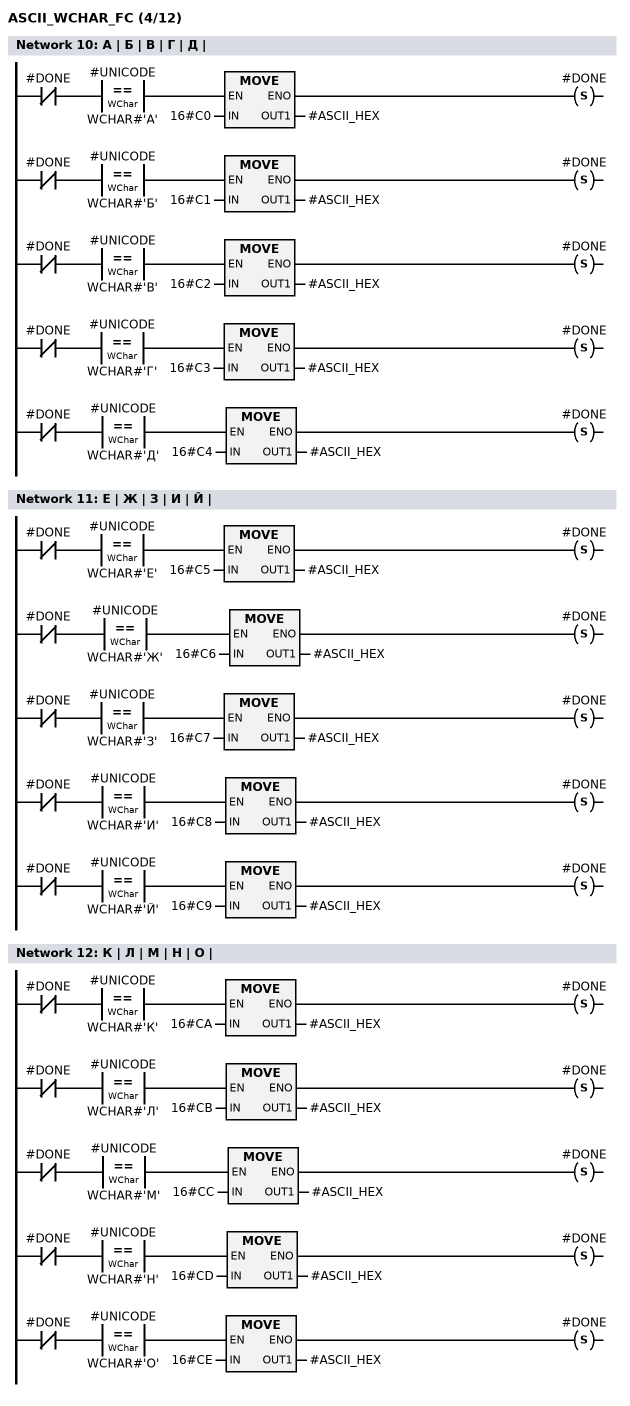
   RUNG wire#powerrail
      I_Contact( #DONE )
      { S7_Templates := "SrcType := WChar" } EQ_Contact(in1 := #UNICODE, in2 := WCHAR#'А')
      Move(in := 16#C0, out1 => #ASCII_HEX)
      S_Coil( #DONE )
   END_RUNG
   RUNG wire#powerrail
      I_Contact( #DONE )
      { S7_Templates := "SrcType := WChar" } EQ_Contact(in1 := #UNICODE, in2 := WCHAR#'Б')
      Move(in := 16#C1, out1 => #ASCII_HEX)
      S_Coil( #DONE )
   END_RUNG
   RUNG wire#powerrail
      I_Contact( #DONE )
      { S7_Templates := "SrcType := WChar" } EQ_Contact(in1 := #UNICODE, in2 := WCHAR#'В')
      Move(in := 16#C2, out1 => #ASCII_HEX)
      S_Coil( #DONE )
   END_RUNG
   RUNG wire#powerrail
      I_Contact( #DONE )
      { S7_Templates := "SrcType := WChar" } EQ_Contact(in1 := #UNICODE, in2 := WCHAR#'Г')
      Move(in := 16#C3, out1 => #ASCII_HEX)
      S_Coil( #DONE )
   END_RUNG
   RUNG wire#powerrail
      I_Contact( #DONE )
      { S7_Templates := "SrcType := WChar" } EQ_Contact(in1 := #UNICODE, in2 := WCHAR#'Д')
      Move(in := 16#C4, out1 => #ASCII_HEX)
      S_Coil( #DONE )
   END_RUNG
   // the same network as SCL:
   IF NOT #DONE AND (#UNICODE = WCHAR#'А') THEN
       #ASCII_HEX := 16#C0;
       #DONE := TRUE;
   END_IF;
   IF NOT #DONE AND (#UNICODE = WCHAR#'Б') THEN
       #ASCII_HEX := 16#C1;
       #DONE := TRUE;
   END_IF;
   IF NOT #DONE AND (#UNICODE = WCHAR#'В') THEN
       #ASCII_HEX := 16#C2;
       #DONE := TRUE;
   END_IF;
   IF NOT #DONE AND (#UNICODE = WCHAR#'Г') THEN
       #ASCII_HEX := 16#C3;
       #DONE := TRUE;
   END_IF;
   IF NOT #DONE AND (#UNICODE = WCHAR#'Д') THEN
       #ASCII_HEX := 16#C4;
       #DONE := TRUE;
   END_IF;
END_REGION

REGION Network 11: Е | Ж | З | И | Й |
   RUNG wire#powerrail
      I_Contact( #DONE )
      { S7_Templates := "SrcType := WChar" } EQ_Contact(in1 := #UNICODE, in2 := WCHAR#'Е')
      Move(in := 16#C5, out1 => #ASCII_HEX)
      S_Coil( #DONE )
   END_RUNG
   RUNG wire#powerrail
      I_Contact( #DONE )
      { S7_Templates := "SrcType := WChar" } EQ_Contact(in1 := #UNICODE, in2 := WCHAR#'Ж')
      Move(in := 16#C6, out1 => #ASCII_HEX)
      S_Coil( #DONE )
   END_RUNG
   RUNG wire#powerrail
      I_Contact( #DONE )
      { S7_Templates := "SrcType := WChar" } EQ_Contact(in1 := #UNICODE, in2 := WCHAR#'З')
      Move(in := 16#C7, out1 => #ASCII_HEX)
      S_Coil( #DONE )
   END_RUNG
   RUNG wire#powerrail
      I_Contact( #DONE )
      { S7_Templates := "SrcType := WChar" } EQ_Contact(in1 := #UNICODE, in2 := WCHAR#'И')
      Move(in := 16#C8, out1 => #ASCII_HEX)
      S_Coil( #DONE )
   END_RUNG
   RUNG wire#powerrail
      I_Contact( #DONE )
      { S7_Templates := "SrcType := WChar" } EQ_Contact(in1 := #UNICODE, in2 := WCHAR#'Й')
      Move(in := 16#C9, out1 => #ASCII_HEX)
      S_Coil( #DONE )
   END_RUNG
   // the same network as SCL:
   IF NOT #DONE AND (#UNICODE = WCHAR#'Е') THEN
       #ASCII_HEX := 16#C5;
       #DONE := TRUE;
   END_IF;
   IF NOT #DONE AND (#UNICODE = WCHAR#'Ж') THEN
       #ASCII_HEX := 16#C6;
       #DONE := TRUE;
   END_IF;
   IF NOT #DONE AND (#UNICODE = WCHAR#'З') THEN
       #ASCII_HEX := 16#C7;
       #DONE := TRUE;
   END_IF;
   IF NOT #DONE AND (#UNICODE = WCHAR#'И') THEN
       #ASCII_HEX := 16#C8;
       #DONE := TRUE;
   END_IF;
   IF NOT #DONE AND (#UNICODE = WCHAR#'Й') THEN
       #ASCII_HEX := 16#C9;
       #DONE := TRUE;
   END_IF;
END_REGION

REGION Network 12: К | Л | М | Н | О |
   RUNG wire#powerrail
      I_Contact( #DONE )
      { S7_Templates := "SrcType := WChar" } EQ_Contact(in1 := #UNICODE, in2 := WCHAR#'К')
      Move(in := 16#CA, out1 => #ASCII_HEX)
      S_Coil( #DONE )
   END_RUNG
   RUNG wire#powerrail
      I_Contact( #DONE )
      { S7_Templates := "SrcType := WChar" } EQ_Contact(in1 := #UNICODE, in2 := WCHAR#'Л')
      Move(in := 16#CB, out1 => #ASCII_HEX)
      S_Coil( #DONE )
   END_RUNG
   RUNG wire#powerrail
      I_Contact( #DONE )
      { S7_Templates := "SrcType := WChar" } EQ_Contact(in1 := #UNICODE, in2 := WCHAR#'М')
      Move(in := 16#CC, out1 => #ASCII_HEX)
      S_Coil( #DONE )
   END_RUNG
   RUNG wire#powerrail
      I_Contact( #DONE )
      { S7_Templates := "SrcType := WChar" } EQ_Contact(in1 := #UNICODE, in2 := WCHAR#'Н')
      Move(in := 16#CD, out1 => #ASCII_HEX)
      S_Coil( #DONE )
   END_RUNG
   RUNG wire#powerrail
      I_Contact( #DONE )
      { S7_Templates := "SrcType := WChar" } EQ_Contact(in1 := #UNICODE, in2 := WCHAR#'О')
      Move(in := 16#CE, out1 => #ASCII_HEX)
      S_Coil( #DONE )
   END_RUNG
   // the same network as SCL:
   IF NOT #DONE AND (#UNICODE = WCHAR#'К') THEN
       #ASCII_HEX := 16#CA;
       #DONE := TRUE;
   END_IF;
   IF NOT #DONE AND (#UNICODE = WCHAR#'Л') THEN
       #ASCII_HEX := 16#CB;
       #DONE := TRUE;
   END_IF;
   IF NOT #DONE AND (#UNICODE = WCHAR#'М') THEN
       #ASCII_HEX := 16#CC;
       #DONE := TRUE;
   END_IF;
   IF NOT #DONE AND (#UNICODE = WCHAR#'Н') THEN
       #ASCII_HEX := 16#CD;
       #DONE := TRUE;
   END_IF;
   IF NOT #DONE AND (#UNICODE = WCHAR#'О') THEN
       #ASCII_HEX := 16#CE;
       #DONE := TRUE;
   END_IF;
END_REGION

REGION Network 13: П | Р | С | Т | У |
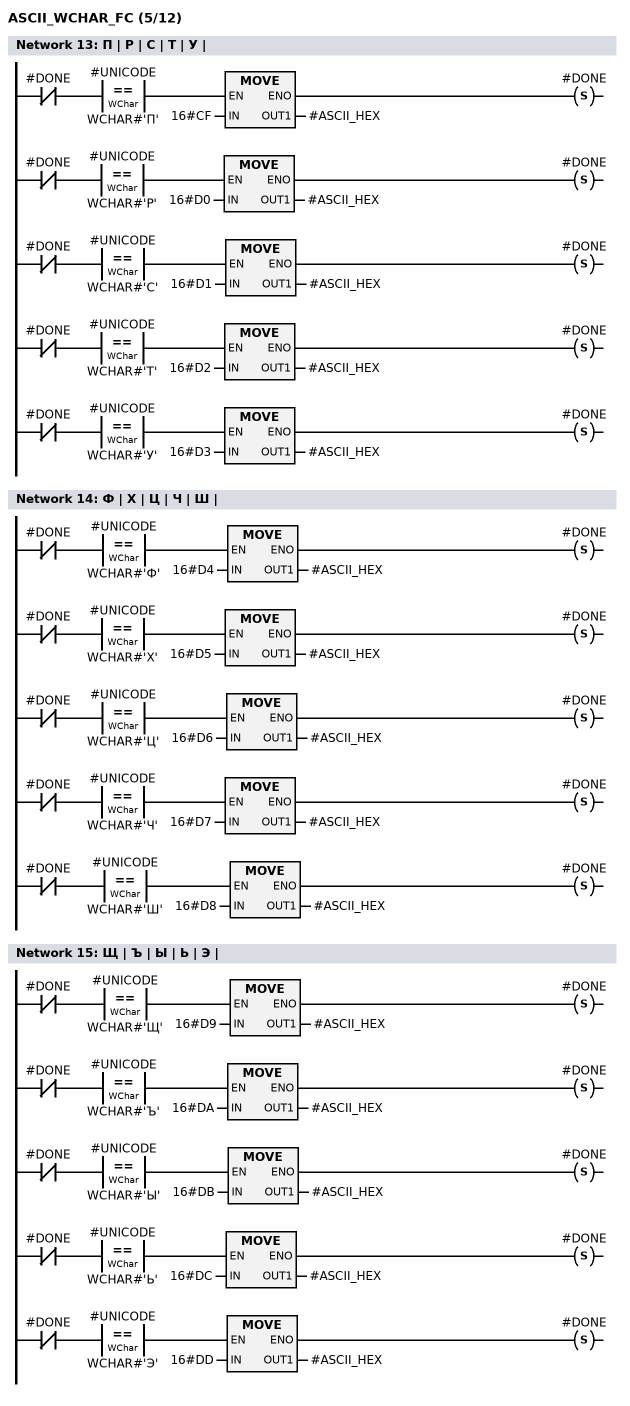
   RUNG wire#powerrail
      I_Contact( #DONE )
      { S7_Templates := "SrcType := WChar" } EQ_Contact(in1 := #UNICODE, in2 := WCHAR#'П')
      Move(in := 16#CF, out1 => #ASCII_HEX)
      S_Coil( #DONE )
   END_RUNG
   RUNG wire#powerrail
      I_Contact( #DONE )
      { S7_Templates := "SrcType := WChar" } EQ_Contact(in1 := #UNICODE, in2 := WCHAR#'Р')
      Move(in := 16#D0, out1 => #ASCII_HEX)
      S_Coil( #DONE )
   END_RUNG
   RUNG wire#powerrail
      I_Contact( #DONE )
      { S7_Templates := "SrcType := WChar" } EQ_Contact(in1 := #UNICODE, in2 := WCHAR#'С')
      Move(in := 16#D1, out1 => #ASCII_HEX)
      S_Coil( #DONE )
   END_RUNG
   RUNG wire#powerrail
      I_Contact( #DONE )
      { S7_Templates := "SrcType := WChar" } EQ_Contact(in1 := #UNICODE, in2 := WCHAR#'Т')
      Move(in := 16#D2, out1 => #ASCII_HEX)
      S_Coil( #DONE )
   END_RUNG
   RUNG wire#powerrail
      I_Contact( #DONE )
      { S7_Templates := "SrcType := WChar" } EQ_Contact(in1 := #UNICODE, in2 := WCHAR#'У')
      Move(in := 16#D3, out1 => #ASCII_HEX)
      S_Coil( #DONE )
   END_RUNG
   // the same network as SCL:
   IF NOT #DONE AND (#UNICODE = WCHAR#'П') THEN
       #ASCII_HEX := 16#CF;
       #DONE := TRUE;
   END_IF;
   IF NOT #DONE AND (#UNICODE = WCHAR#'Р') THEN
       #ASCII_HEX := 16#D0;
       #DONE := TRUE;
   END_IF;
   IF NOT #DONE AND (#UNICODE = WCHAR#'С') THEN
       #ASCII_HEX := 16#D1;
       #DONE := TRUE;
   END_IF;
   IF NOT #DONE AND (#UNICODE = WCHAR#'Т') THEN
       #ASCII_HEX := 16#D2;
       #DONE := TRUE;
   END_IF;
   IF NOT #DONE AND (#UNICODE = WCHAR#'У') THEN
       #ASCII_HEX := 16#D3;
       #DONE := TRUE;
   END_IF;
END_REGION

REGION Network 14: Ф | Х | Ц | Ч | Ш |
   RUNG wire#powerrail
      I_Contact( #DONE )
      { S7_Templates := "SrcType := WChar" } EQ_Contact(in1 := #UNICODE, in2 := WCHAR#'Ф')
      Move(in := 16#D4, out1 => #ASCII_HEX)
      S_Coil( #DONE )
   END_RUNG
   RUNG wire#powerrail
      I_Contact( #DONE )
      { S7_Templates := "SrcType := WChar" } EQ_Contact(in1 := #UNICODE, in2 := WCHAR#'Х')
      Move(in := 16#D5, out1 => #ASCII_HEX)
      S_Coil( #DONE )
   END_RUNG
   RUNG wire#powerrail
      I_Contact( #DONE )
      { S7_Templates := "SrcType := WChar" } EQ_Contact(in1 := #UNICODE, in2 := WCHAR#'Ц')
      Move(in := 16#D6, out1 => #ASCII_HEX)
      S_Coil( #DONE )
   END_RUNG
   RUNG wire#powerrail
      I_Contact( #DONE )
      { S7_Templates := "SrcType := WChar" } EQ_Contact(in1 := #UNICODE, in2 := WCHAR#'Ч')
      Move(in := 16#D7, out1 => #ASCII_HEX)
      S_Coil( #DONE )
   END_RUNG
   RUNG wire#powerrail
      I_Contact( #DONE )
      { S7_Templates := "SrcType := WChar" } EQ_Contact(in1 := #UNICODE, in2 := WCHAR#'Ш')
      Move(in := 16#D8, out1 => #ASCII_HEX)
      S_Coil( #DONE )
   END_RUNG
   // the same network as SCL:
   IF NOT #DONE AND (#UNICODE = WCHAR#'Ф') THEN
       #ASCII_HEX := 16#D4;
       #DONE := TRUE;
   END_IF;
   IF NOT #DONE AND (#UNICODE = WCHAR#'Х') THEN
       #ASCII_HEX := 16#D5;
       #DONE := TRUE;
   END_IF;
   IF NOT #DONE AND (#UNICODE = WCHAR#'Ц') THEN
       #ASCII_HEX := 16#D6;
       #DONE := TRUE;
   END_IF;
   IF NOT #DONE AND (#UNICODE = WCHAR#'Ч') THEN
       #ASCII_HEX := 16#D7;
       #DONE := TRUE;
   END_IF;
   IF NOT #DONE AND (#UNICODE = WCHAR#'Ш') THEN
       #ASCII_HEX := 16#D8;
       #DONE := TRUE;
   END_IF;
END_REGION

REGION Network 15: Щ | Ъ | Ы | Ь | Э |
   RUNG wire#powerrail
      I_Contact( #DONE )
      { S7_Templates := "SrcType := WChar" } EQ_Contact(in1 := #UNICODE, in2 := WCHAR#'Щ')
      Move(in := 16#D9, out1 => #ASCII_HEX)
      S_Coil( #DONE )
   END_RUNG
   RUNG wire#powerrail
      I_Contact( #DONE )
      { S7_Templates := "SrcType := WChar" } EQ_Contact(in1 := #UNICODE, in2 := WCHAR#'Ъ')
      Move(in := 16#DA, out1 => #ASCII_HEX)
      S_Coil( #DONE )
   END_RUNG
   RUNG wire#powerrail
      I_Contact( #DONE )
      { S7_Templates := "SrcType := WChar" } EQ_Contact(in1 := #UNICODE, in2 := WCHAR#'Ы')
      Move(in := 16#DB, out1 => #ASCII_HEX)
      S_Coil( #DONE )
   END_RUNG
   RUNG wire#powerrail
      I_Contact( #DONE )
      { S7_Templates := "SrcType := WChar" } EQ_Contact(in1 := #UNICODE, in2 := WCHAR#'Ь')
      Move(in := 16#DC, out1 => #ASCII_HEX)
      S_Coil( #DONE )
   END_RUNG
   RUNG wire#powerrail
      I_Contact( #DONE )
      { S7_Templates := "SrcType := WChar" } EQ_Contact(in1 := #UNICODE, in2 := WCHAR#'Э')
      Move(in := 16#DD, out1 => #ASCII_HEX)
      S_Coil( #DONE )
   END_RUNG
   // the same network as SCL:
   IF NOT #DONE AND (#UNICODE = WCHAR#'Щ') THEN
       #ASCII_HEX := 16#D9;
       #DONE := TRUE;
   END_IF;
   IF NOT #DONE AND (#UNICODE = WCHAR#'Ъ') THEN
       #ASCII_HEX := 16#DA;
       #DONE := TRUE;
   END_IF;
   IF NOT #DONE AND (#UNICODE = WCHAR#'Ы') THEN
       #ASCII_HEX := 16#DB;
       #DONE := TRUE;
   END_IF;
   IF NOT #DONE AND (#UNICODE = WCHAR#'Ь') THEN
       #ASCII_HEX := 16#DC;
       #DONE := TRUE;
   END_IF;
   IF NOT #DONE AND (#UNICODE = WCHAR#'Э') THEN
       #ASCII_HEX := 16#DD;
       #DONE := TRUE;
   END_IF;
END_REGION

REGION Network 16: Ю | Я |
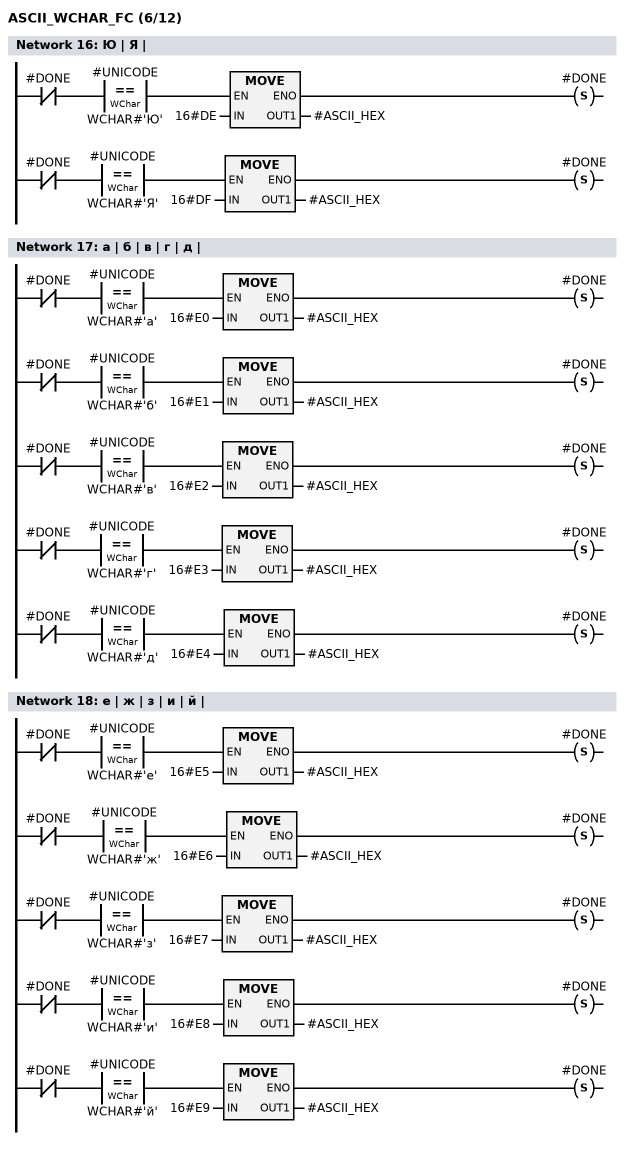
   RUNG wire#powerrail
      I_Contact( #DONE )
      { S7_Templates := "SrcType := WChar" } EQ_Contact(in1 := #UNICODE, in2 := WCHAR#'Ю')
      Move(in := 16#DE, out1 => #ASCII_HEX)
      S_Coil( #DONE )
   END_RUNG
   RUNG wire#powerrail
      I_Contact( #DONE )
      { S7_Templates := "SrcType := WChar" } EQ_Contact(in1 := #UNICODE, in2 := WCHAR#'Я')
      Move(in := 16#DF, out1 => #ASCII_HEX)
      S_Coil( #DONE )
   END_RUNG
   // the same network as SCL:
   IF NOT #DONE AND (#UNICODE = WCHAR#'Ю') THEN
       #ASCII_HEX := 16#DE;
       #DONE := TRUE;
   END_IF;
   IF NOT #DONE AND (#UNICODE = WCHAR#'Я') THEN
       #ASCII_HEX := 16#DF;
       #DONE := TRUE;
   END_IF;
END_REGION

REGION Network 17: а | б | в | г | д |
   RUNG wire#powerrail
      I_Contact( #DONE )
      { S7_Templates := "SrcType := WChar" } EQ_Contact(in1 := #UNICODE, in2 := WCHAR#'а')
      Move(in := 16#E0, out1 => #ASCII_HEX)
      S_Coil( #DONE )
   END_RUNG
   RUNG wire#powerrail
      I_Contact( #DONE )
      { S7_Templates := "SrcType := WChar" } EQ_Contact(in1 := #UNICODE, in2 := WCHAR#'б')
      Move(in := 16#E1, out1 => #ASCII_HEX)
      S_Coil( #DONE )
   END_RUNG
   RUNG wire#powerrail
      I_Contact( #DONE )
      { S7_Templates := "SrcType := WChar" } EQ_Contact(in1 := #UNICODE, in2 := WCHAR#'в')
      Move(in := 16#E2, out1 => #ASCII_HEX)
      S_Coil( #DONE )
   END_RUNG
   RUNG wire#powerrail
      I_Contact( #DONE )
      { S7_Templates := "SrcType := WChar" } EQ_Contact(in1 := #UNICODE, in2 := WCHAR#'г')
      Move(in := 16#E3, out1 => #ASCII_HEX)
      S_Coil( #DONE )
   END_RUNG
   RUNG wire#powerrail
      I_Contact( #DONE )
      { S7_Templates := "SrcType := WChar" } EQ_Contact(in1 := #UNICODE, in2 := WCHAR#'д')
      Move(in := 16#E4, out1 => #ASCII_HEX)
      S_Coil( #DONE )
   END_RUNG
   // the same network as SCL:
   IF NOT #DONE AND (#UNICODE = WCHAR#'а') THEN
       #ASCII_HEX := 16#E0;
       #DONE := TRUE;
   END_IF;
   IF NOT #DONE AND (#UNICODE = WCHAR#'б') THEN
       #ASCII_HEX := 16#E1;
       #DONE := TRUE;
   END_IF;
   IF NOT #DONE AND (#UNICODE = WCHAR#'в') THEN
       #ASCII_HEX := 16#E2;
       #DONE := TRUE;
   END_IF;
   IF NOT #DONE AND (#UNICODE = WCHAR#'г') THEN
       #ASCII_HEX := 16#E3;
       #DONE := TRUE;
   END_IF;
   IF NOT #DONE AND (#UNICODE = WCHAR#'д') THEN
       #ASCII_HEX := 16#E4;
       #DONE := TRUE;
   END_IF;
END_REGION

REGION Network 18: е | ж | з | и | й |
   RUNG wire#powerrail
      I_Contact( #DONE )
      { S7_Templates := "SrcType := WChar" } EQ_Contact(in1 := #UNICODE, in2 := WCHAR#'е')
      Move(in := 16#E5, out1 => #ASCII_HEX)
      S_Coil( #DONE )
   END_RUNG
   RUNG wire#powerrail
      I_Contact( #DONE )
      { S7_Templates := "SrcType := WChar" } EQ_Contact(in1 := #UNICODE, in2 := WCHAR#'ж')
      Move(in := 16#E6, out1 => #ASCII_HEX)
      S_Coil( #DONE )
   END_RUNG
   RUNG wire#powerrail
      I_Contact( #DONE )
      { S7_Templates := "SrcType := WChar" } EQ_Contact(in1 := #UNICODE, in2 := WCHAR#'з')
      Move(in := 16#E7, out1 => #ASCII_HEX)
      S_Coil( #DONE )
   END_RUNG
   RUNG wire#powerrail
      I_Contact( #DONE )
      { S7_Templates := "SrcType := WChar" } EQ_Contact(in1 := #UNICODE, in2 := WCHAR#'и')
      Move(in := 16#E8, out1 => #ASCII_HEX)
      S_Coil( #DONE )
   END_RUNG
   RUNG wire#powerrail
      I_Contact( #DONE )
      { S7_Templates := "SrcType := WChar" } EQ_Contact(in1 := #UNICODE, in2 := WCHAR#'й')
      Move(in := 16#E9, out1 => #ASCII_HEX)
      S_Coil( #DONE )
   END_RUNG
   // the same network as SCL:
   IF NOT #DONE AND (#UNICODE = WCHAR#'е') THEN
       #ASCII_HEX := 16#E5;
       #DONE := TRUE;
   END_IF;
   IF NOT #DONE AND (#UNICODE = WCHAR#'ж') THEN
       #ASCII_HEX := 16#E6;
       #DONE := TRUE;
   END_IF;
   IF NOT #DONE AND (#UNICODE = WCHAR#'з') THEN
       #ASCII_HEX := 16#E7;
       #DONE := TRUE;
   END_IF;
   IF NOT #DONE AND (#UNICODE = WCHAR#'и') THEN
       #ASCII_HEX := 16#E8;
       #DONE := TRUE;
   END_IF;
   IF NOT #DONE AND (#UNICODE = WCHAR#'й') THEN
       #ASCII_HEX := 16#E9;
       #DONE := TRUE;
   END_IF;
END_REGION

REGION Network 19: к | л | м | н | о |
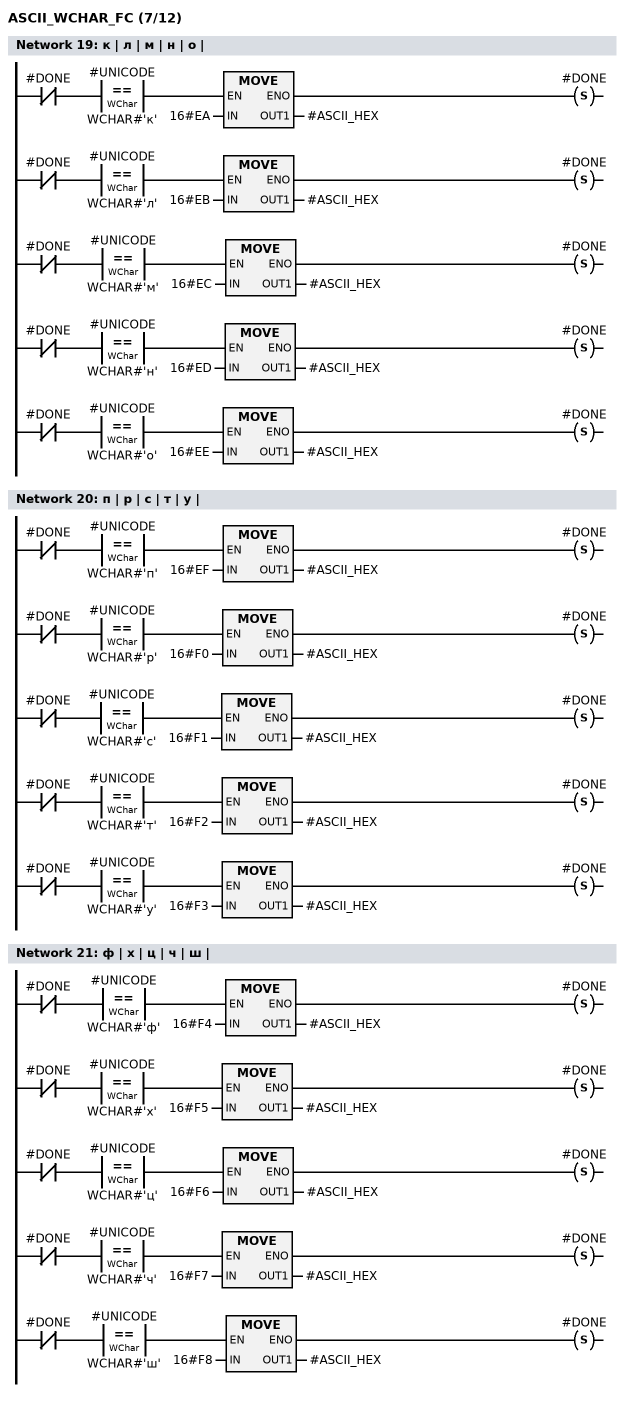
   RUNG wire#powerrail
      I_Contact( #DONE )
      { S7_Templates := "SrcType := WChar" } EQ_Contact(in1 := #UNICODE, in2 := WCHAR#'к')
      Move(in := 16#EA, out1 => #ASCII_HEX)
      S_Coil( #DONE )
   END_RUNG
   RUNG wire#powerrail
      I_Contact( #DONE )
      { S7_Templates := "SrcType := WChar" } EQ_Contact(in1 := #UNICODE, in2 := WCHAR#'л')
      Move(in := 16#EB, out1 => #ASCII_HEX)
      S_Coil( #DONE )
   END_RUNG
   RUNG wire#powerrail
      I_Contact( #DONE )
      { S7_Templates := "SrcType := WChar" } EQ_Contact(in1 := #UNICODE, in2 := WCHAR#'м')
      Move(in := 16#EC, out1 => #ASCII_HEX)
      S_Coil( #DONE )
   END_RUNG
   RUNG wire#powerrail
      I_Contact( #DONE )
      { S7_Templates := "SrcType := WChar" } EQ_Contact(in1 := #UNICODE, in2 := WCHAR#'н')
      Move(in := 16#ED, out1 => #ASCII_HEX)
      S_Coil( #DONE )
   END_RUNG
   RUNG wire#powerrail
      I_Contact( #DONE )
      { S7_Templates := "SrcType := WChar" } EQ_Contact(in1 := #UNICODE, in2 := WCHAR#'о')
      Move(in := 16#EE, out1 => #ASCII_HEX)
      S_Coil( #DONE )
   END_RUNG
   // the same network as SCL:
   IF NOT #DONE AND (#UNICODE = WCHAR#'к') THEN
       #ASCII_HEX := 16#EA;
       #DONE := TRUE;
   END_IF;
   IF NOT #DONE AND (#UNICODE = WCHAR#'л') THEN
       #ASCII_HEX := 16#EB;
       #DONE := TRUE;
   END_IF;
   IF NOT #DONE AND (#UNICODE = WCHAR#'м') THEN
       #ASCII_HEX := 16#EC;
       #DONE := TRUE;
   END_IF;
   IF NOT #DONE AND (#UNICODE = WCHAR#'н') THEN
       #ASCII_HEX := 16#ED;
       #DONE := TRUE;
   END_IF;
   IF NOT #DONE AND (#UNICODE = WCHAR#'о') THEN
       #ASCII_HEX := 16#EE;
       #DONE := TRUE;
   END_IF;
END_REGION

REGION Network 20: п | р | с | т | у |
   RUNG wire#powerrail
      I_Contact( #DONE )
      { S7_Templates := "SrcType := WChar" } EQ_Contact(in1 := #UNICODE, in2 := WCHAR#'п')
      Move(in := 16#EF, out1 => #ASCII_HEX)
      S_Coil( #DONE )
   END_RUNG
   RUNG wire#powerrail
      I_Contact( #DONE )
      { S7_Templates := "SrcType := WChar" } EQ_Contact(in1 := #UNICODE, in2 := WCHAR#'р')
      Move(in := 16#F0, out1 => #ASCII_HEX)
      S_Coil( #DONE )
   END_RUNG
   RUNG wire#powerrail
      I_Contact( #DONE )
      { S7_Templates := "SrcType := WChar" } EQ_Contact(in1 := #UNICODE, in2 := WCHAR#'с')
      Move(in := 16#F1, out1 => #ASCII_HEX)
      S_Coil( #DONE )
   END_RUNG
   RUNG wire#powerrail
      I_Contact( #DONE )
      { S7_Templates := "SrcType := WChar" } EQ_Contact(in1 := #UNICODE, in2 := WCHAR#'т')
      Move(in := 16#F2, out1 => #ASCII_HEX)
      S_Coil( #DONE )
   END_RUNG
   RUNG wire#powerrail
      I_Contact( #DONE )
      { S7_Templates := "SrcType := WChar" } EQ_Contact(in1 := #UNICODE, in2 := WCHAR#'у')
      Move(in := 16#F3, out1 => #ASCII_HEX)
      S_Coil( #DONE )
   END_RUNG
   // the same network as SCL:
   IF NOT #DONE AND (#UNICODE = WCHAR#'п') THEN
       #ASCII_HEX := 16#EF;
       #DONE := TRUE;
   END_IF;
   IF NOT #DONE AND (#UNICODE = WCHAR#'р') THEN
       #ASCII_HEX := 16#F0;
       #DONE := TRUE;
   END_IF;
   IF NOT #DONE AND (#UNICODE = WCHAR#'с') THEN
       #ASCII_HEX := 16#F1;
       #DONE := TRUE;
   END_IF;
   IF NOT #DONE AND (#UNICODE = WCHAR#'т') THEN
       #ASCII_HEX := 16#F2;
       #DONE := TRUE;
   END_IF;
   IF NOT #DONE AND (#UNICODE = WCHAR#'у') THEN
       #ASCII_HEX := 16#F3;
       #DONE := TRUE;
   END_IF;
END_REGION

REGION Network 21: ф | х | ц | ч | ш |
   RUNG wire#powerrail
      I_Contact( #DONE )
      { S7_Templates := "SrcType := WChar" } EQ_Contact(in1 := #UNICODE, in2 := WCHAR#'ф')
      Move(in := 16#F4, out1 => #ASCII_HEX)
      S_Coil( #DONE )
   END_RUNG
   RUNG wire#powerrail
      I_Contact( #DONE )
      { S7_Templates := "SrcType := WChar" } EQ_Contact(in1 := #UNICODE, in2 := WCHAR#'х')
      Move(in := 16#F5, out1 => #ASCII_HEX)
      S_Coil( #DONE )
   END_RUNG
   RUNG wire#powerrail
      I_Contact( #DONE )
      { S7_Templates := "SrcType := WChar" } EQ_Contact(in1 := #UNICODE, in2 := WCHAR#'ц')
      Move(in := 16#F6, out1 => #ASCII_HEX)
      S_Coil( #DONE )
   END_RUNG
   RUNG wire#powerrail
      I_Contact( #DONE )
      { S7_Templates := "SrcType := WChar" } EQ_Contact(in1 := #UNICODE, in2 := WCHAR#'ч')
      Move(in := 16#F7, out1 => #ASCII_HEX)
      S_Coil( #DONE )
   END_RUNG
   RUNG wire#powerrail
      I_Contact( #DONE )
      { S7_Templates := "SrcType := WChar" } EQ_Contact(in1 := #UNICODE, in2 := WCHAR#'ш')
      Move(in := 16#F8, out1 => #ASCII_HEX)
      S_Coil( #DONE )
   END_RUNG
   // the same network as SCL:
   IF NOT #DONE AND (#UNICODE = WCHAR#'ф') THEN
       #ASCII_HEX := 16#F4;
       #DONE := TRUE;
   END_IF;
   IF NOT #DONE AND (#UNICODE = WCHAR#'х') THEN
       #ASCII_HEX := 16#F5;
       #DONE := TRUE;
   END_IF;
   IF NOT #DONE AND (#UNICODE = WCHAR#'ц') THEN
       #ASCII_HEX := 16#F6;
       #DONE := TRUE;
   END_IF;
   IF NOT #DONE AND (#UNICODE = WCHAR#'ч') THEN
       #ASCII_HEX := 16#F7;
       #DONE := TRUE;
   END_IF;
   IF NOT #DONE AND (#UNICODE = WCHAR#'ш') THEN
       #ASCII_HEX := 16#F8;
       #DONE := TRUE;
   END_IF;
END_REGION

REGION Network 22: щ | ъ | ы | ь | э |
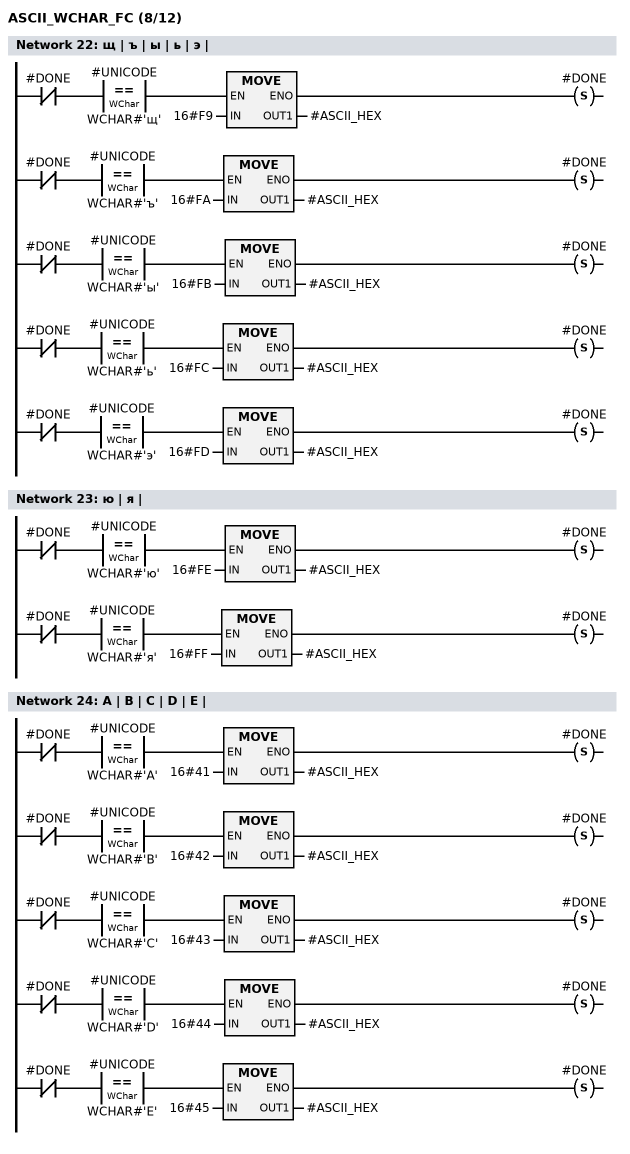
   RUNG wire#powerrail
      I_Contact( #DONE )
      { S7_Templates := "SrcType := WChar" } EQ_Contact(in1 := #UNICODE, in2 := WCHAR#'щ')
      Move(in := 16#F9, out1 => #ASCII_HEX)
      S_Coil( #DONE )
   END_RUNG
   RUNG wire#powerrail
      I_Contact( #DONE )
      { S7_Templates := "SrcType := WChar" } EQ_Contact(in1 := #UNICODE, in2 := WCHAR#'ъ')
      Move(in := 16#FA, out1 => #ASCII_HEX)
      S_Coil( #DONE )
   END_RUNG
   RUNG wire#powerrail
      I_Contact( #DONE )
      { S7_Templates := "SrcType := WChar" } EQ_Contact(in1 := #UNICODE, in2 := WCHAR#'ы')
      Move(in := 16#FB, out1 => #ASCII_HEX)
      S_Coil( #DONE )
   END_RUNG
   RUNG wire#powerrail
      I_Contact( #DONE )
      { S7_Templates := "SrcType := WChar" } EQ_Contact(in1 := #UNICODE, in2 := WCHAR#'ь')
      Move(in := 16#FC, out1 => #ASCII_HEX)
      S_Coil( #DONE )
   END_RUNG
   RUNG wire#powerrail
      I_Contact( #DONE )
      { S7_Templates := "SrcType := WChar" } EQ_Contact(in1 := #UNICODE, in2 := WCHAR#'э')
      Move(in := 16#FD, out1 => #ASCII_HEX)
      S_Coil( #DONE )
   END_RUNG
   // the same network as SCL:
   IF NOT #DONE AND (#UNICODE = WCHAR#'щ') THEN
       #ASCII_HEX := 16#F9;
       #DONE := TRUE;
   END_IF;
   IF NOT #DONE AND (#UNICODE = WCHAR#'ъ') THEN
       #ASCII_HEX := 16#FA;
       #DONE := TRUE;
   END_IF;
   IF NOT #DONE AND (#UNICODE = WCHAR#'ы') THEN
       #ASCII_HEX := 16#FB;
       #DONE := TRUE;
   END_IF;
   IF NOT #DONE AND (#UNICODE = WCHAR#'ь') THEN
       #ASCII_HEX := 16#FC;
       #DONE := TRUE;
   END_IF;
   IF NOT #DONE AND (#UNICODE = WCHAR#'э') THEN
       #ASCII_HEX := 16#FD;
       #DONE := TRUE;
   END_IF;
END_REGION

REGION Network 23: ю | я |
   RUNG wire#powerrail
      I_Contact( #DONE )
      { S7_Templates := "SrcType := WChar" } EQ_Contact(in1 := #UNICODE, in2 := WCHAR#'ю')
      Move(in := 16#FE, out1 => #ASCII_HEX)
      S_Coil( #DONE )
   END_RUNG
   RUNG wire#powerrail
      I_Contact( #DONE )
      { S7_Templates := "SrcType := WChar" } EQ_Contact(in1 := #UNICODE, in2 := WCHAR#'я')
      Move(in := 16#FF, out1 => #ASCII_HEX)
      S_Coil( #DONE )
   END_RUNG
   // the same network as SCL:
   IF NOT #DONE AND (#UNICODE = WCHAR#'ю') THEN
       #ASCII_HEX := 16#FE;
       #DONE := TRUE;
   END_IF;
   IF NOT #DONE AND (#UNICODE = WCHAR#'я') THEN
       #ASCII_HEX := 16#FF;
       #DONE := TRUE;
   END_IF;
END_REGION

REGION Network 24: A | B | C | D | E |
   RUNG wire#powerrail
      I_Contact( #DONE )
      { S7_Templates := "SrcType := WChar" } EQ_Contact(in1 := #UNICODE, in2 := WCHAR#'A')
      Move(in := 16#41, out1 => #ASCII_HEX)
      S_Coil( #DONE )
   END_RUNG
   RUNG wire#powerrail
      I_Contact( #DONE )
      { S7_Templates := "SrcType := WChar" } EQ_Contact(in1 := #UNICODE, in2 := WCHAR#'B')
      Move(in := 16#42, out1 => #ASCII_HEX)
      S_Coil( #DONE )
   END_RUNG
   RUNG wire#powerrail
      I_Contact( #DONE )
      { S7_Templates := "SrcType := WChar" } EQ_Contact(in1 := #UNICODE, in2 := WCHAR#'C')
      Move(in := 16#43, out1 => #ASCII_HEX)
      S_Coil( #DONE )
   END_RUNG
   RUNG wire#powerrail
      I_Contact( #DONE )
      { S7_Templates := "SrcType := WChar" } EQ_Contact(in1 := #UNICODE, in2 := WCHAR#'D')
      Move(in := 16#44, out1 => #ASCII_HEX)
      S_Coil( #DONE )
   END_RUNG
   RUNG wire#powerrail
      I_Contact( #DONE )
      { S7_Templates := "SrcType := WChar" } EQ_Contact(in1 := #UNICODE, in2 := WCHAR#'E')
      Move(in := 16#45, out1 => #ASCII_HEX)
      S_Coil( #DONE )
   END_RUNG
   // the same network as SCL:
   IF NOT #DONE AND (#UNICODE = WCHAR#'A') THEN
       #ASCII_HEX := 16#41;
       #DONE := TRUE;
   END_IF;
   IF NOT #DONE AND (#UNICODE = WCHAR#'B') THEN
       #ASCII_HEX := 16#42;
       #DONE := TRUE;
   END_IF;
   IF NOT #DONE AND (#UNICODE = WCHAR#'C') THEN
       #ASCII_HEX := 16#43;
       #DONE := TRUE;
   END_IF;
   IF NOT #DONE AND (#UNICODE = WCHAR#'D') THEN
       #ASCII_HEX := 16#44;
       #DONE := TRUE;
   END_IF;
   IF NOT #DONE AND (#UNICODE = WCHAR#'E') THEN
       #ASCII_HEX := 16#45;
       #DONE := TRUE;
   END_IF;
END_REGION

REGION Network 25: F | G | H | I | J |
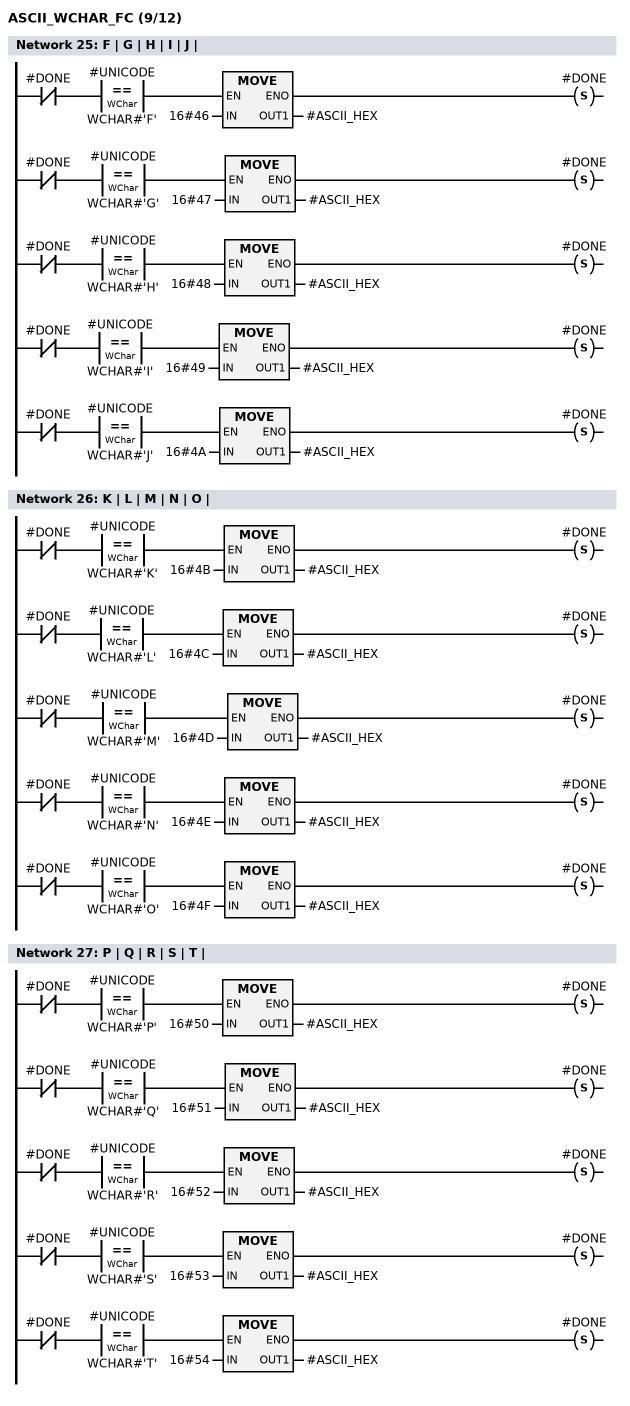
   RUNG wire#powerrail
      I_Contact( #DONE )
      { S7_Templates := "SrcType := WChar" } EQ_Contact(in1 := #UNICODE, in2 := WCHAR#'F')
      Move(in := 16#46, out1 => #ASCII_HEX)
      S_Coil( #DONE )
   END_RUNG
   RUNG wire#powerrail
      I_Contact( #DONE )
      { S7_Templates := "SrcType := WChar" } EQ_Contact(in1 := #UNICODE, in2 := WCHAR#'G')
      Move(in := 16#47, out1 => #ASCII_HEX)
      S_Coil( #DONE )
   END_RUNG
   RUNG wire#powerrail
      I_Contact( #DONE )
      { S7_Templates := "SrcType := WChar" } EQ_Contact(in1 := #UNICODE, in2 := WCHAR#'H')
      Move(in := 16#48, out1 => #ASCII_HEX)
      S_Coil( #DONE )
   END_RUNG
   RUNG wire#powerrail
      I_Contact( #DONE )
      { S7_Templates := "SrcType := WChar" } EQ_Contact(in1 := #UNICODE, in2 := WCHAR#'I')
      Move(in := 16#49, out1 => #ASCII_HEX)
      S_Coil( #DONE )
   END_RUNG
   RUNG wire#powerrail
      I_Contact( #DONE )
      { S7_Templates := "SrcType := WChar" } EQ_Contact(in1 := #UNICODE, in2 := WCHAR#'J')
      Move(in := 16#4A, out1 => #ASCII_HEX)
      S_Coil( #DONE )
   END_RUNG
   // the same network as SCL:
   IF NOT #DONE AND (#UNICODE = WCHAR#'F') THEN
       #ASCII_HEX := 16#46;
       #DONE := TRUE;
   END_IF;
   IF NOT #DONE AND (#UNICODE = WCHAR#'G') THEN
       #ASCII_HEX := 16#47;
       #DONE := TRUE;
   END_IF;
   IF NOT #DONE AND (#UNICODE = WCHAR#'H') THEN
       #ASCII_HEX := 16#48;
       #DONE := TRUE;
   END_IF;
   IF NOT #DONE AND (#UNICODE = WCHAR#'I') THEN
       #ASCII_HEX := 16#49;
       #DONE := TRUE;
   END_IF;
   IF NOT #DONE AND (#UNICODE = WCHAR#'J') THEN
       #ASCII_HEX := 16#4A;
       #DONE := TRUE;
   END_IF;
END_REGION

REGION Network 26: K | L | M | N | O |
   RUNG wire#powerrail
      I_Contact( #DONE )
      { S7_Templates := "SrcType := WChar" } EQ_Contact(in1 := #UNICODE, in2 := WCHAR#'K')
      Move(in := 16#4B, out1 => #ASCII_HEX)
      S_Coil( #DONE )
   END_RUNG
   RUNG wire#powerrail
      I_Contact( #DONE )
      { S7_Templates := "SrcType := WChar" } EQ_Contact(in1 := #UNICODE, in2 := WCHAR#'L')
      Move(in := 16#4C, out1 => #ASCII_HEX)
      S_Coil( #DONE )
   END_RUNG
   RUNG wire#powerrail
      I_Contact( #DONE )
      { S7_Templates := "SrcType := WChar" } EQ_Contact(in1 := #UNICODE, in2 := WCHAR#'M')
      Move(in := 16#4D, out1 => #ASCII_HEX)
      S_Coil( #DONE )
   END_RUNG
   RUNG wire#powerrail
      I_Contact( #DONE )
      { S7_Templates := "SrcType := WChar" } EQ_Contact(in1 := #UNICODE, in2 := WCHAR#'N')
      Move(in := 16#4E, out1 => #ASCII_HEX)
      S_Coil( #DONE )
   END_RUNG
   RUNG wire#powerrail
      I_Contact( #DONE )
      { S7_Templates := "SrcType := WChar" } EQ_Contact(in1 := #UNICODE, in2 := WCHAR#'O')
      Move(in := 16#4F, out1 => #ASCII_HEX)
      S_Coil( #DONE )
   END_RUNG
   // the same network as SCL:
   IF NOT #DONE AND (#UNICODE = WCHAR#'K') THEN
       #ASCII_HEX := 16#4B;
       #DONE := TRUE;
   END_IF;
   IF NOT #DONE AND (#UNICODE = WCHAR#'L') THEN
       #ASCII_HEX := 16#4C;
       #DONE := TRUE;
   END_IF;
   IF NOT #DONE AND (#UNICODE = WCHAR#'M') THEN
       #ASCII_HEX := 16#4D;
       #DONE := TRUE;
   END_IF;
   IF NOT #DONE AND (#UNICODE = WCHAR#'N') THEN
       #ASCII_HEX := 16#4E;
       #DONE := TRUE;
   END_IF;
   IF NOT #DONE AND (#UNICODE = WCHAR#'O') THEN
       #ASCII_HEX := 16#4F;
       #DONE := TRUE;
   END_IF;
END_REGION

REGION Network 27: P | Q | R | S | T |
   RUNG wire#powerrail
      I_Contact( #DONE )
      { S7_Templates := "SrcType := WChar" } EQ_Contact(in1 := #UNICODE, in2 := WCHAR#'P')
      Move(in := 16#50, out1 => #ASCII_HEX)
      S_Coil( #DONE )
   END_RUNG
   RUNG wire#powerrail
      I_Contact( #DONE )
      { S7_Templates := "SrcType := WChar" } EQ_Contact(in1 := #UNICODE, in2 := WCHAR#'Q')
      Move(in := 16#51, out1 => #ASCII_HEX)
      S_Coil( #DONE )
   END_RUNG
   RUNG wire#powerrail
      I_Contact( #DONE )
      { S7_Templates := "SrcType := WChar" } EQ_Contact(in1 := #UNICODE, in2 := WCHAR#'R')
      Move(in := 16#52, out1 => #ASCII_HEX)
      S_Coil( #DONE )
   END_RUNG
   RUNG wire#powerrail
      I_Contact( #DONE )
      { S7_Templates := "SrcType := WChar" } EQ_Contact(in1 := #UNICODE, in2 := WCHAR#'S')
      Move(in := 16#53, out1 => #ASCII_HEX)
      S_Coil( #DONE )
   END_RUNG
   RUNG wire#powerrail
      I_Contact( #DONE )
      { S7_Templates := "SrcType := WChar" } EQ_Contact(in1 := #UNICODE, in2 := WCHAR#'T')
      Move(in := 16#54, out1 => #ASCII_HEX)
      S_Coil( #DONE )
   END_RUNG
   // the same network as SCL:
   IF NOT #DONE AND (#UNICODE = WCHAR#'P') THEN
       #ASCII_HEX := 16#50;
       #DONE := TRUE;
   END_IF;
   IF NOT #DONE AND (#UNICODE = WCHAR#'Q') THEN
       #ASCII_HEX := 16#51;
       #DONE := TRUE;
   END_IF;
   IF NOT #DONE AND (#UNICODE = WCHAR#'R') THEN
       #ASCII_HEX := 16#52;
       #DONE := TRUE;
   END_IF;
   IF NOT #DONE AND (#UNICODE = WCHAR#'S') THEN
       #ASCII_HEX := 16#53;
       #DONE := TRUE;
   END_IF;
   IF NOT #DONE AND (#UNICODE = WCHAR#'T') THEN
       #ASCII_HEX := 16#54;
       #DONE := TRUE;
   END_IF;
END_REGION

REGION Network 28: U | V | W | X | Y | Z |
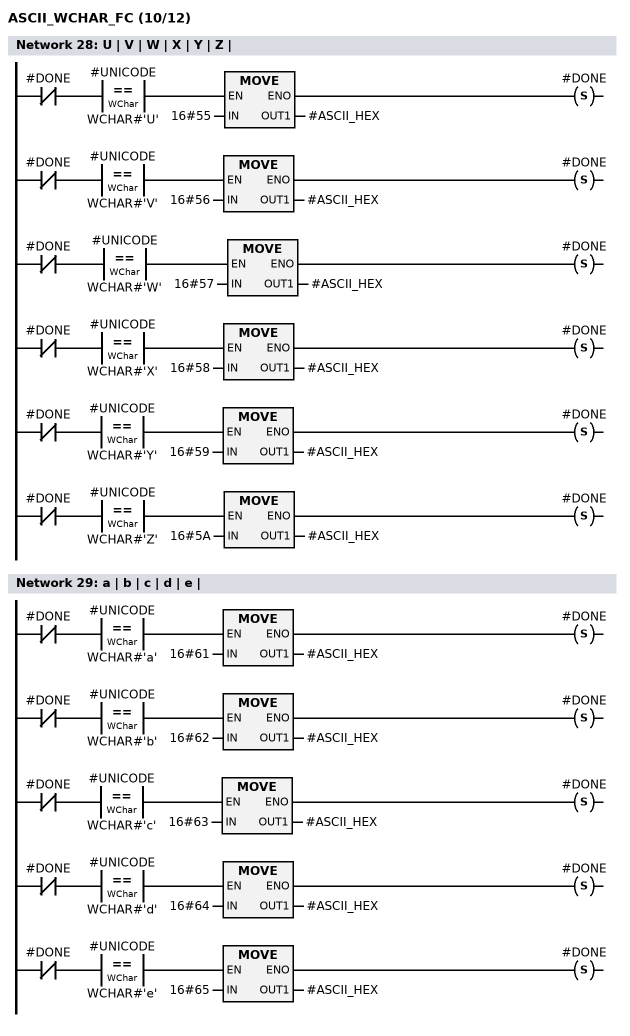
   RUNG wire#powerrail
      I_Contact( #DONE )
      { S7_Templates := "SrcType := WChar" } EQ_Contact(in1 := #UNICODE, in2 := WCHAR#'U')
      Move(in := 16#55, out1 => #ASCII_HEX)
      S_Coil( #DONE )
   END_RUNG
   RUNG wire#powerrail
      I_Contact( #DONE )
      { S7_Templates := "SrcType := WChar" } EQ_Contact(in1 := #UNICODE, in2 := WCHAR#'V')
      Move(in := 16#56, out1 => #ASCII_HEX)
      S_Coil( #DONE )
   END_RUNG
   RUNG wire#powerrail
      I_Contact( #DONE )
      { S7_Templates := "SrcType := WChar" } EQ_Contact(in1 := #UNICODE, in2 := WCHAR#'W')
      Move(in := 16#57, out1 => #ASCII_HEX)
      S_Coil( #DONE )
   END_RUNG
   RUNG wire#powerrail
      I_Contact( #DONE )
      { S7_Templates := "SrcType := WChar" } EQ_Contact(in1 := #UNICODE, in2 := WCHAR#'X')
      Move(in := 16#58, out1 => #ASCII_HEX)
      S_Coil( #DONE )
   END_RUNG
   RUNG wire#powerrail
      I_Contact( #DONE )
      { S7_Templates := "SrcType := WChar" } EQ_Contact(in1 := #UNICODE, in2 := WCHAR#'Y')
      Move(in := 16#59, out1 => #ASCII_HEX)
      S_Coil( #DONE )
   END_RUNG
   RUNG wire#powerrail
      I_Contact( #DONE )
      { S7_Templates := "SrcType := WChar" } EQ_Contact(in1 := #UNICODE, in2 := WCHAR#'Z')
      Move(in := 16#5A, out1 => #ASCII_HEX)
      S_Coil( #DONE )
   END_RUNG
   // the same network as SCL:
   IF NOT #DONE AND (#UNICODE = WCHAR#'U') THEN
       #ASCII_HEX := 16#55;
       #DONE := TRUE;
   END_IF;
   IF NOT #DONE AND (#UNICODE = WCHAR#'V') THEN
       #ASCII_HEX := 16#56;
       #DONE := TRUE;
   END_IF;
   IF NOT #DONE AND (#UNICODE = WCHAR#'W') THEN
       #ASCII_HEX := 16#57;
       #DONE := TRUE;
   END_IF;
   IF NOT #DONE AND (#UNICODE = WCHAR#'X') THEN
       #ASCII_HEX := 16#58;
       #DONE := TRUE;
   END_IF;
   IF NOT #DONE AND (#UNICODE = WCHAR#'Y') THEN
       #ASCII_HEX := 16#59;
       #DONE := TRUE;
   END_IF;
   IF NOT #DONE AND (#UNICODE = WCHAR#'Z') THEN
       #ASCII_HEX := 16#5A;
       #DONE := TRUE;
   END_IF;
END_REGION

REGION Network 29: a | b | c | d | e |
   RUNG wire#powerrail
      I_Contact( #DONE )
      { S7_Templates := "SrcType := WChar" } EQ_Contact(in1 := #UNICODE, in2 := WCHAR#'a')
      Move(in := 16#61, out1 => #ASCII_HEX)
      S_Coil( #DONE )
   END_RUNG
   RUNG wire#powerrail
      I_Contact( #DONE )
      { S7_Templates := "SrcType := WChar" } EQ_Contact(in1 := #UNICODE, in2 := WCHAR#'b')
      Move(in := 16#62, out1 => #ASCII_HEX)
      S_Coil( #DONE )
   END_RUNG
   RUNG wire#powerrail
      I_Contact( #DONE )
      { S7_Templates := "SrcType := WChar" } EQ_Contact(in1 := #UNICODE, in2 := WCHAR#'c')
      Move(in := 16#63, out1 => #ASCII_HEX)
      S_Coil( #DONE )
   END_RUNG
   RUNG wire#powerrail
      I_Contact( #DONE )
      { S7_Templates := "SrcType := WChar" } EQ_Contact(in1 := #UNICODE, in2 := WCHAR#'d')
      Move(in := 16#64, out1 => #ASCII_HEX)
      S_Coil( #DONE )
   END_RUNG
   RUNG wire#powerrail
      I_Contact( #DONE )
      { S7_Templates := "SrcType := WChar" } EQ_Contact(in1 := #UNICODE, in2 := WCHAR#'e')
      Move(in := 16#65, out1 => #ASCII_HEX)
      S_Coil( #DONE )
   END_RUNG
   // the same network as SCL:
   IF NOT #DONE AND (#UNICODE = WCHAR#'a') THEN
       #ASCII_HEX := 16#61;
       #DONE := TRUE;
   END_IF;
   IF NOT #DONE AND (#UNICODE = WCHAR#'b') THEN
       #ASCII_HEX := 16#62;
       #DONE := TRUE;
   END_IF;
   IF NOT #DONE AND (#UNICODE = WCHAR#'c') THEN
       #ASCII_HEX := 16#63;
       #DONE := TRUE;
   END_IF;
   IF NOT #DONE AND (#UNICODE = WCHAR#'d') THEN
       #ASCII_HEX := 16#64;
       #DONE := TRUE;
   END_IF;
   IF NOT #DONE AND (#UNICODE = WCHAR#'e') THEN
       #ASCII_HEX := 16#65;
       #DONE := TRUE;
   END_IF;
END_REGION

REGION Network 30: f | g | h | i | j |
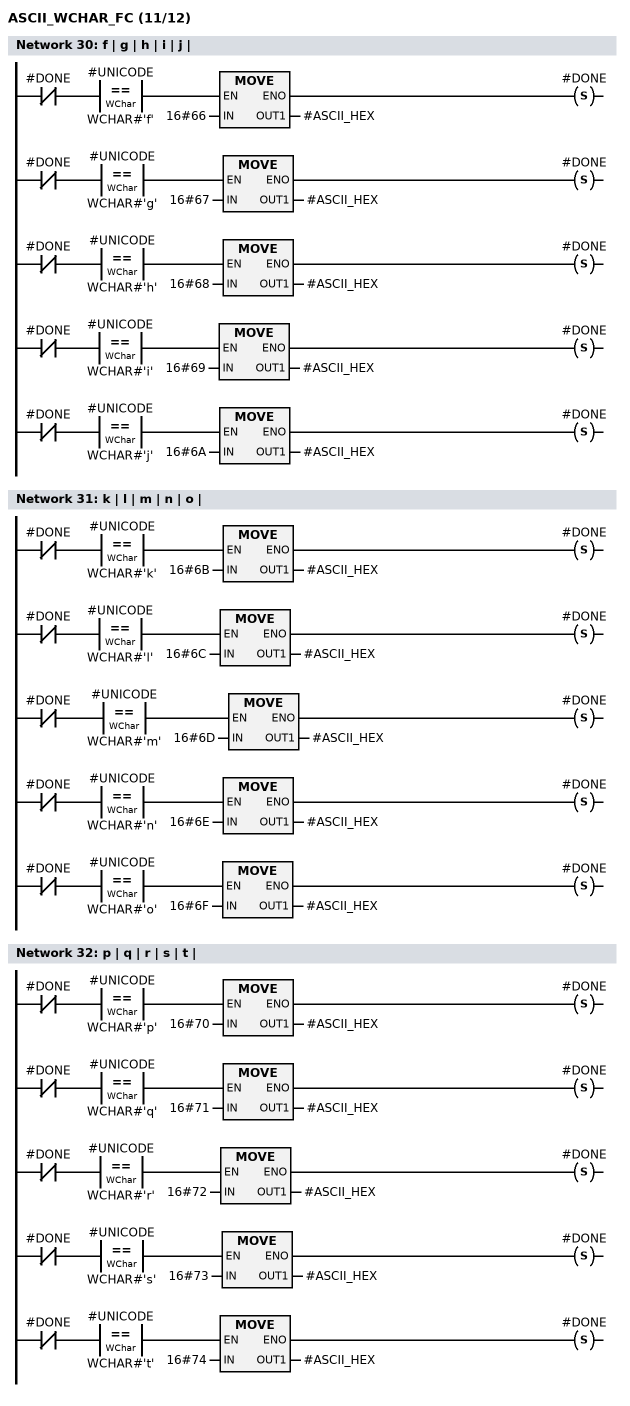
   RUNG wire#powerrail
      I_Contact( #DONE )
      { S7_Templates := "SrcType := WChar" } EQ_Contact(in1 := #UNICODE, in2 := WCHAR#'f')
      Move(in := 16#66, out1 => #ASCII_HEX)
      S_Coil( #DONE )
   END_RUNG
   RUNG wire#powerrail
      I_Contact( #DONE )
      { S7_Templates := "SrcType := WChar" } EQ_Contact(in1 := #UNICODE, in2 := WCHAR#'g')
      Move(in := 16#67, out1 => #ASCII_HEX)
      S_Coil( #DONE )
   END_RUNG
   RUNG wire#powerrail
      I_Contact( #DONE )
      { S7_Templates := "SrcType := WChar" } EQ_Contact(in1 := #UNICODE, in2 := WCHAR#'h')
      Move(in := 16#68, out1 => #ASCII_HEX)
      S_Coil( #DONE )
   END_RUNG
   RUNG wire#powerrail
      I_Contact( #DONE )
      { S7_Templates := "SrcType := WChar" } EQ_Contact(in1 := #UNICODE, in2 := WCHAR#'i')
      Move(in := 16#69, out1 => #ASCII_HEX)
      S_Coil( #DONE )
   END_RUNG
   RUNG wire#powerrail
      I_Contact( #DONE )
      { S7_Templates := "SrcType := WChar" } EQ_Contact(in1 := #UNICODE, in2 := WCHAR#'j')
      Move(in := 16#6A, out1 => #ASCII_HEX)
      S_Coil( #DONE )
   END_RUNG
   // the same network as SCL:
   IF NOT #DONE AND (#UNICODE = WCHAR#'f') THEN
       #ASCII_HEX := 16#66;
       #DONE := TRUE;
   END_IF;
   IF NOT #DONE AND (#UNICODE = WCHAR#'g') THEN
       #ASCII_HEX := 16#67;
       #DONE := TRUE;
   END_IF;
   IF NOT #DONE AND (#UNICODE = WCHAR#'h') THEN
       #ASCII_HEX := 16#68;
       #DONE := TRUE;
   END_IF;
   IF NOT #DONE AND (#UNICODE = WCHAR#'i') THEN
       #ASCII_HEX := 16#69;
       #DONE := TRUE;
   END_IF;
   IF NOT #DONE AND (#UNICODE = WCHAR#'j') THEN
       #ASCII_HEX := 16#6A;
       #DONE := TRUE;
   END_IF;
END_REGION

REGION Network 31: k | l | m | n | o |
   RUNG wire#powerrail
      I_Contact( #DONE )
      { S7_Templates := "SrcType := WChar" } EQ_Contact(in1 := #UNICODE, in2 := WCHAR#'k')
      Move(in := 16#6B, out1 => #ASCII_HEX)
      S_Coil( #DONE )
   END_RUNG
   RUNG wire#powerrail
      I_Contact( #DONE )
      { S7_Templates := "SrcType := WChar" } EQ_Contact(in1 := #UNICODE, in2 := WCHAR#'l')
      Move(in := 16#6C, out1 => #ASCII_HEX)
      S_Coil( #DONE )
   END_RUNG
   RUNG wire#powerrail
      I_Contact( #DONE )
      { S7_Templates := "SrcType := WChar" } EQ_Contact(in1 := #UNICODE, in2 := WCHAR#'m')
      Move(in := 16#6D, out1 => #ASCII_HEX)
      S_Coil( #DONE )
   END_RUNG
   RUNG wire#powerrail
      I_Contact( #DONE )
      { S7_Templates := "SrcType := WChar" } EQ_Contact(in1 := #UNICODE, in2 := WCHAR#'n')
      Move(in := 16#6E, out1 => #ASCII_HEX)
      S_Coil( #DONE )
   END_RUNG
   RUNG wire#powerrail
      I_Contact( #DONE )
      { S7_Templates := "SrcType := WChar" } EQ_Contact(in1 := #UNICODE, in2 := WCHAR#'o')
      Move(in := 16#6F, out1 => #ASCII_HEX)
      S_Coil( #DONE )
   END_RUNG
   // the same network as SCL:
   IF NOT #DONE AND (#UNICODE = WCHAR#'k') THEN
       #ASCII_HEX := 16#6B;
       #DONE := TRUE;
   END_IF;
   IF NOT #DONE AND (#UNICODE = WCHAR#'l') THEN
       #ASCII_HEX := 16#6C;
       #DONE := TRUE;
   END_IF;
   IF NOT #DONE AND (#UNICODE = WCHAR#'m') THEN
       #ASCII_HEX := 16#6D;
       #DONE := TRUE;
   END_IF;
   IF NOT #DONE AND (#UNICODE = WCHAR#'n') THEN
       #ASCII_HEX := 16#6E;
       #DONE := TRUE;
   END_IF;
   IF NOT #DONE AND (#UNICODE = WCHAR#'o') THEN
       #ASCII_HEX := 16#6F;
       #DONE := TRUE;
   END_IF;
END_REGION

REGION Network 32: p | q | r | s | t |
   RUNG wire#powerrail
      I_Contact( #DONE )
      { S7_Templates := "SrcType := WChar" } EQ_Contact(in1 := #UNICODE, in2 := WCHAR#'p')
      Move(in := 16#70, out1 => #ASCII_HEX)
      S_Coil( #DONE )
   END_RUNG
   RUNG wire#powerrail
      I_Contact( #DONE )
      { S7_Templates := "SrcType := WChar" } EQ_Contact(in1 := #UNICODE, in2 := WCHAR#'q')
      Move(in := 16#71, out1 => #ASCII_HEX)
      S_Coil( #DONE )
   END_RUNG
   RUNG wire#powerrail
      I_Contact( #DONE )
      { S7_Templates := "SrcType := WChar" } EQ_Contact(in1 := #UNICODE, in2 := WCHAR#'r')
      Move(in := 16#72, out1 => #ASCII_HEX)
      S_Coil( #DONE )
   END_RUNG
   RUNG wire#powerrail
      I_Contact( #DONE )
      { S7_Templates := "SrcType := WChar" } EQ_Contact(in1 := #UNICODE, in2 := WCHAR#'s')
      Move(in := 16#73, out1 => #ASCII_HEX)
      S_Coil( #DONE )
   END_RUNG
   RUNG wire#powerrail
      I_Contact( #DONE )
      { S7_Templates := "SrcType := WChar" } EQ_Contact(in1 := #UNICODE, in2 := WCHAR#'t')
      Move(in := 16#74, out1 => #ASCII_HEX)
      S_Coil( #DONE )
   END_RUNG
   // the same network as SCL:
   IF NOT #DONE AND (#UNICODE = WCHAR#'p') THEN
       #ASCII_HEX := 16#70;
       #DONE := TRUE;
   END_IF;
   IF NOT #DONE AND (#UNICODE = WCHAR#'q') THEN
       #ASCII_HEX := 16#71;
       #DONE := TRUE;
   END_IF;
   IF NOT #DONE AND (#UNICODE = WCHAR#'r') THEN
       #ASCII_HEX := 16#72;
       #DONE := TRUE;
   END_IF;
   IF NOT #DONE AND (#UNICODE = WCHAR#'s') THEN
       #ASCII_HEX := 16#73;
       #DONE := TRUE;
   END_IF;
   IF NOT #DONE AND (#UNICODE = WCHAR#'t') THEN
       #ASCII_HEX := 16#74;
       #DONE := TRUE;
   END_IF;
END_REGION

REGION Network 33: u | v | w | x | y | z |
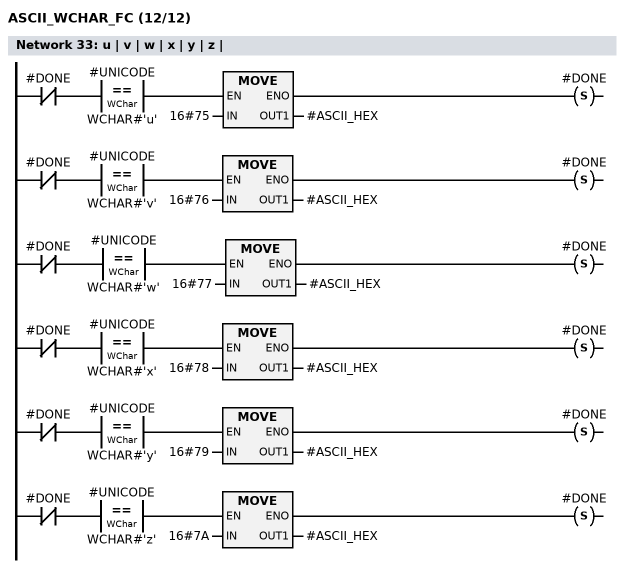
   RUNG wire#powerrail
      I_Contact( #DONE )
      { S7_Templates := "SrcType := WChar" } EQ_Contact(in1 := #UNICODE, in2 := WCHAR#'u')
      Move(in := 16#75, out1 => #ASCII_HEX)
      S_Coil( #DONE )
   END_RUNG
   RUNG wire#powerrail
      I_Contact( #DONE )
      { S7_Templates := "SrcType := WChar" } EQ_Contact(in1 := #UNICODE, in2 := WCHAR#'v')
      Move(in := 16#76, out1 => #ASCII_HEX)
      S_Coil( #DONE )
   END_RUNG
   RUNG wire#powerrail
      I_Contact( #DONE )
      { S7_Templates := "SrcType := WChar" } EQ_Contact(in1 := #UNICODE, in2 := WCHAR#'w')
      Move(in := 16#77, out1 => #ASCII_HEX)
      S_Coil( #DONE )
   END_RUNG
   RUNG wire#powerrail
      I_Contact( #DONE )
      { S7_Templates := "SrcType := WChar" } EQ_Contact(in1 := #UNICODE, in2 := WCHAR#'x')
      Move(in := 16#78, out1 => #ASCII_HEX)
      S_Coil( #DONE )
   END_RUNG
   RUNG wire#powerrail
      I_Contact( #DONE )
      { S7_Templates := "SrcType := WChar" } EQ_Contact(in1 := #UNICODE, in2 := WCHAR#'y')
      Move(in := 16#79, out1 => #ASCII_HEX)
      S_Coil( #DONE )
   END_RUNG
   RUNG wire#powerrail
      I_Contact( #DONE )
      { S7_Templates := "SrcType := WChar" } EQ_Contact(in1 := #UNICODE, in2 := WCHAR#'z')
      Move(in := 16#7A, out1 => #ASCII_HEX)
      S_Coil( #DONE )
   END_RUNG
   // the same network as SCL:
   IF NOT #DONE AND (#UNICODE = WCHAR#'u') THEN
       #ASCII_HEX := 16#75;
       #DONE := TRUE;
   END_IF;
   IF NOT #DONE AND (#UNICODE = WCHAR#'v') THEN
       #ASCII_HEX := 16#76;
       #DONE := TRUE;
   END_IF;
   IF NOT #DONE AND (#UNICODE = WCHAR#'w') THEN
       #ASCII_HEX := 16#77;
       #DONE := TRUE;
   END_IF;
   IF NOT #DONE AND (#UNICODE = WCHAR#'x') THEN
       #ASCII_HEX := 16#78;
       #DONE := TRUE;
   END_IF;
   IF NOT #DONE AND (#UNICODE = WCHAR#'y') THEN
       #ASCII_HEX := 16#79;
       #DONE := TRUE;
   END_IF;
   IF NOT #DONE AND (#UNICODE = WCHAR#'z') THEN
       #ASCII_HEX := 16#7A;
       #DONE := TRUE;
   END_IF;
END_REGION
END_FUNCTION

DATA_BLOCK "Gaz_status_DB"   // DB3
VERSION : 0.1
// stored: AutoNumber true, DBAccessibleFromOPCUA true, InstanceOfName Gaz_status, InstanceOfType FB
"Gaz_status"
BEGIN
END_DATA_BLOCK

DATA_BLOCK "Line_Control_DB"   // DB5
VERSION : 0.1
// stored: AutoNumber false, DBAccessibleFromOPCUA true, InstanceOfName Line_Control, InstanceOfType FB
"Line_Control"
BEGIN
   Line[0..2].Hand := FALSE;
   Line[0..2].SP_Source := TRUE;
   Line[0..2].PID_Not_Use := FALSE;
   Line[0..2].Mode := FALSE;
   Line[0..2].RM_1_Report_DI := FALSE;
   Line[0..2].RM_2_Report_DI := FALSE;
   Line[0..2].RM_Weight := 1.0;
   Line[0].SP_M := 0.0;
   Line[1].SP_M := 1.0;
   Line[2].SP_M := 0.0;
   Line[0..2].SP_min := 10.0;
   Line[0..2].SP_max := 200.0;
   Line[0..2].PE_min := 0.15;
   Line[0..2].PE_max := 2.5;
   Line[0..2].D := 0.0;
   Line[0..2].C_Tank := 0.0;
   Line[0..2].Low_Flow := 0.0;
   Line[0].Res_SP := 0.0;
   Line[1].Res_SP := 4.0;
   Line[2].Res_SP := 0.0;
   Line[0..2].Use.RT := FALSE;
   Line[0..2].Use.RM := FALSE;
   Line[0..2].Use.SP := TRUE;
   Line[0..2].Use.Flow := FALSE;
   Line[0..2].Use.Res := FALSE;
   Line[0..2].Use.DME := FALSE;
   Line[0..2].Use.PE := FALSE;
   Line[0..2].PID.CMD.Vector := FALSE;
   Line[0..2].PID.x := 1.0;
   Line[0..2].PID.Settings.SP_P := 1.5;
   Line[0..2].PID.Settings.SP_Ti := 150.0;
   Line[0..2].PID.Settings.SP_Td := 0.0;
   Line[0..2].PID.Settings.SP_Cycle := 0.2;
   Line[0..2].PID.Settings.Max_SP := 500.0;
   Line[0..2].PID.Settings.Min_SP := -500.0;
   Line[0..2].PID.Settings.Max_in := 500.0;
   Line[0..2].PID.Settings.Min_in := -500.0;
   Line[0..2].PID.Settings.Max_out := 100.0;
   Line[0..2].PID.Settings.Min_out := 0.0;
   Line[0].PID.Settings.DeadBand := 0.0;
   Line[1..2].PID.Settings.DeadBand := 1.0;
   Line[0..2].PID.PID.IntegralResetMode := 4;
   Line[0..2].PID.PID.RunModeByStartup := TRUE;
   Line[0..2].PID.PID.SetSubstituteOutput := TRUE;
   Line[0..2].PID.PID.ActivateRecoverMode := TRUE;
   Line[0..2].PID.PID.CancelTuningLevel := 10.0;
   Line[0..2].PID.PID.SubstituteOutput := 0.0;
   Line[0].PID.PID.Config.InputPerOn := TRUE;
   Line[1..2].PID.PID.Config.InputPerOn := FALSE;
   Line[0..2].PID.PID.Config.InvertControl := FALSE;
   Line[0].PID.PID.Config.InputUpperLimit := 120.0;
   Line[1..2].PID.PID.Config.InputUpperLimit := 500.0;
   Line[0].PID.PID.Config.InputLowerLimit := 0.0;
   Line[1..2].PID.PID.Config.InputLowerLimit := -500.0;
   Line[0..2].PID.PID.Config.InputUpperWarning := 3.402822E+38;
   Line[0..2].PID.PID.Config.InputLowerWarning := -3.402822E+38;
   Line[0..2].PID.PID.Config.OutputUpperLimit := 100.0;
   Line[0..2].PID.PID.Config.OutputLowerLimit := 0.0;
   Line[0].PID.PID.Config.SetpointUpperLimit := 3.402822E+38;
   Line[1..2].PID.PID.Config.SetpointUpperLimit := 500.0;
   Line[0].PID.PID.Config.SetpointLowerLimit := -3.402822E+38;
   Line[1..2].PID.PID.Config.SetpointLowerLimit := -500.0;
   Line[0..2].PID.PID.Config.MinimumOnTime := 0.0;
   Line[0..2].PID.PID.Config.MinimumOffTime := 0.0;
   Line[0..2].PID.PID.Config.InputScaling.UpperPointIn := 27648.0;
   Line[0..2].PID.PID.Config.InputScaling.LowerPointIn := 0.0;
   Line[0..2].PID.PID.Config.InputScaling.UpperPointOut := 100.0;
   Line[0..2].PID.PID.Config.InputScaling.LowerPointOut := 0.0;
   Line[0..2].PID.PID.CycleTime.EnEstimation := TRUE;
   Line[0..2].PID.PID.CycleTime.EnMonitoring := TRUE;
   Line[0].PID.PID.CycleTime.Value := 0.1;
   Line[1].PID.PID.CycleTime.Value := 0.2005259;
   Line[2].PID.PID.CycleTime.Value := 0.2005263;
   Line[0..2].PID.PID.CtrlParamsBackUp.Gain := 1.0;
   Line[0..2].PID.PID.CtrlParamsBackUp.Ti := 20.0;
   Line[0..2].PID.PID.CtrlParamsBackUp.Td := 0.0;
   Line[0..2].PID.PID.CtrlParamsBackUp.TdFiltRatio := 0.2;
   Line[0..2].PID.PID.CtrlParamsBackUp.PWeighting := 1.0;
   Line[0..2].PID.PID.CtrlParamsBackUp.DWeighting := 1.0;
   Line[0..2].PID.PID.CtrlParamsBackUp.Cycle := 1.0;
   Line[0].PID.PID.PIDSelfTune.SUT.TuneRule := 0;
   Line[1..2].PID.PID.PIDSelfTune.SUT.TuneRule := 1;
   Line[0..2].PID.PID.PIDSelfTune.TIR.TuneRule := 0;
   Line[0].PID.PID.Retain.CtrlParams.Gain := 1.0;
   Line[1..2].PID.PID.Retain.CtrlParams.Gain := 1.5;
   Line[0].PID.PID.Retain.CtrlParams.Ti := 20.0;
   Line[1..2].PID.PID.Retain.CtrlParams.Ti := 150.0;
   Line[0..2].PID.PID.Retain.CtrlParams.Td := 0.0;
   Line[0..2].PID.PID.Retain.CtrlParams.TdFiltRatio := 0.2;
   Line[0..2].PID.PID.Retain.CtrlParams.PWeighting := 1.0;
   Line[0..2].PID.PID.Retain.CtrlParams.DWeighting := 1.0;
   Line[0..2].PID.PID.Retain.CtrlParams.Cycle := 1.0;
   Line[0].PID.C.SP := 1.0;
   Line[1..2].PID.C.SP := 0.2;
   Line[0..2].PID.C.One := 0.1;
   Line[0].FlowMeter_1.Mode := FALSE;
   Line[1..2].FlowMeter_1.Mode := TRUE;
   Line[0..2].FlowMeter_1.Fast_Mode := TRUE;
   Line[0..2].FlowMeter_1.clock := 0.01;
   Line[0..2].FlowMeter_1.Weight := 1.0;
   Line[0..2].FlowMeter_1.All := 0.0;
   Line[0..2].FlowMeter_1.Any := 0.0;
   Line[0..2].FlowMeter_1.Seans := 0.0;
   Line[0..2].FlowMeter_1.Seans_Last := 0.0;
   Line[0].FlowMeter_1.Flow_Today := 0.0;
   Line[1..2].FlowMeter_1.Flow_Today := 0.3833334;
   Line[0].FlowMeter_1.Flow_LastDay := 0.0;
   Line[1].FlowMeter_1.Flow_LastDay := 0.3833334;
   Line[2].FlowMeter_1.Flow_LastDay := 0.0;
   Line[0..2].FlowMeter_1.Flow_Lock_All := 0.0;
   Line[0..2].FlowMeter_1.Flow_Lock_Now := 0.0;
   Line[0].FlowMeter_1.ADDR_Byte := 0;
   Line[1].FlowMeter_1.ADDR_Byte := 2;
   Line[2].FlowMeter_1.ADDR_Byte := 0;
   Line[0].FlowMeter_1.ADDR_Bit := 0;
   Line[1].FlowMeter_1.ADDR_Bit := 1;
   Line[2].FlowMeter_1.ADDR_Bit := 0;
   Line[0..2].FlowMeter_1.Filter.Moment := TRUE;
   Line[0].FlowMeter_2.Mode := FALSE;
   Line[1..2].FlowMeter_2.Mode := TRUE;
   Line[0..2].FlowMeter_2.Fast_Mode := TRUE;
   Line[0..2].FlowMeter_2.clock := 0.01;
   Line[0..2].FlowMeter_2.Weight := 1.0;
   Line[0..2].FlowMeter_2.All := 0.0;
   Line[0..2].FlowMeter_2.Any := 0.0;
   Line[0..2].FlowMeter_2.Seans := 0.0;
   Line[0..2].FlowMeter_2.Seans_Last := 0.0;
   Line[0..2].FlowMeter_2.Flow_Today := 0.0;
   Line[0..2].FlowMeter_2.Flow_LastDay := 0.0;
   Line[0..2].FlowMeter_2.Flow_Lock_All := 0.0;
   Line[0..2].FlowMeter_2.Flow_Lock_Now := 0.0;
   Line[0..2].FlowMeter_2.ADDR_Byte := 0;
   Line[0..2].FlowMeter_2.ADDR_Bit := 0;
   Line[0..2].FlowMeter_2.Filter.Moment := TRUE;
   Pump[1..2].Reserv := FALSE;
   Pump[1..2].Line_Main := 1;
   Pump[1..2].Line_Reserv := 0;
END_DATA_BLOCK

DATA_BLOCK "Lock_DB"   // DB2
VERSION : 0.1
// stored: AutoNumber true, DBAccessibleFromOPCUA true, InstanceOfName Lock, InstanceOfType FB
"Lock"
BEGIN
END_DATA_BLOCK

DATA_BLOCK "Logick_DB"   // DB1
VERSION : 0.1
// stored: AutoNumber true, DBAccessibleFromOPCUA true, InstanceOfName Logick, InstanceOfType FB
"Logick"
BEGIN
   ELZ_1.T_Gas.SP_M := 0;
   ELZ_1.T_Gas.SP_S := 30;
   ELZ_1.T_ELZ_Start.SP_M := 0;
   ELZ_1.T_ELZ_Start.SP_S := 5;
   T_Wash.SP_M := 0;
   T_Wash.SP_S := 30;
END_DATA_BLOCK

DATA_BLOCK "ModBus_RTU_DB"   // DB30
VERSION : 0.1
// stored: AutoNumber false, DBAccessibleFromOPCUA true, InstanceOfName ModBus_RTU, InstanceOfType FB
"ModBus_RTU"
BEGIN
   DEV_Config[1..10].Use := FALSE;
   DEV_Config[1..10].MODE := FALSE;
   DEV_Config[1..10].ADDR := 0;
   DEV_Config[1..10].Register := 0;
   DEV_Config[1..10].Length := 0;
   DEV_Config[1..10].Source_DB := 0;
   DEV_Config[1..10].Source_OFFSET := 0;
   DEV_Config[1..10].Target_DB := 0;
   DEV_Config[1..10].Target_OFFSET := 0;
END_DATA_BLOCK

DATA_BLOCK "ModBus_TCP_DB"   // DB40
VERSION : 0.1
// stored: AutoNumber false, DBAccessibleFromOPCUA true, InstanceOfName ModBus_TCP, InstanceOfType FB
"ModBus_TCP"
BEGIN
   CONNECT.InterfaceId := 64;
   CONNECT.ID := 1;
   CONNECT.ConnectionType := 11;
   CONNECT.RemoteAddress.ADDR[1] := 192;
   CONNECT.RemoteAddress.ADDR[2] := 168;
   CONNECT.RemoteAddress.ADDR[3] := 0;
   CONNECT.RemoteAddress.ADDR[4] := 10;
   CONNECT.RemotePort := 502;
END_DATA_BLOCK

DATA_BLOCK "Smena_DB"   // DB26
VERSION : 0.1
// stored: AutoNumber true, DBAccessibleFromOPCUA true, InstanceOfName Smena, InstanceOfType FB
"Smena"
BEGIN
   pos[0..31] := FALSE;
   Line_1[0..2].Water := 0.0;
   Line_1[0..2].Reagent := 0.0;
   Line_2[0..2].Water := 0.0;
   Line_2[0..2].Reagent := 0.0;
   "Time"[0].Start_H := 0;
   "Time"[1].Start_H := 10;
   "Time"[2].Start_H := 6;
   "Time"[0].Start_M := 0;
   "Time"[1].Start_M := 9;
   "Time"[2].Start_M := 0;
   "Time"[0]."Date" := 0;
   "Time"[1..2]."Date" := 10;
   "Time"[0].Mounth := 0;
   "Time"[1].Mounth := 12;
   "Time"[2].Mounth := 9;
END_DATA_BLOCK

DATA_BLOCK "AIx_DB"   // DB220
VERSION : 0.1
// stored: AutoNumber false, DBAccessibleFromOPCUA true, InstanceOfName AIx, InstanceOfType FB
"AIx"
BEGIN
END_DATA_BLOCK

DATA_BLOCK "AOx_DB"   // DB230
VERSION : 0.1
// stored: AutoNumber false, DBAccessibleFromOPCUA true, InstanceOfName AOx, InstanceOfType FB
"AOx"
BEGIN
END_DATA_BLOCK

DATA_BLOCK "DIx_1_DB"   // DB200
VERSION : 0.1
// stored: AutoNumber false, DBAccessibleFromOPCUA true, InstanceOfName DIx_1, InstanceOfType FB
"DIx_1"
BEGIN
   AllBlock.Use.Inverse := TRUE;
   AllBlock.Use.Indirect := TRUE;
   AllBlock.ADDR_Byte := 1;
   AllBlock.ADDR_Bit := 5;
   AllBlock.Filter_On.SP := 16#02;
   AllBlock.Filter_Off.SP := 16#02;
   EZ_1_FB_AHLS.Use.Inverse := TRUE;
   EZ_1_FB_AHLS.Use.Indirect := TRUE;
   EZ_1_FB_AHLS.ADDR_Byte := 2;
   EZ_1_FB_AHLS.ADDR_Bit := 2;
   EZ_1_FB_AHLS.Filter_On.SP := 16#02;
   EZ_1_FB_AHLS.Filter_Off.SP := 16#02;
   Gas_Chanel_1_1.Use.Inverse := TRUE;
   Gas_Chanel_1_1.Use.Indirect := TRUE;
   Gas_Chanel_1_1.ADDR_Byte := 0;
   Gas_Chanel_1_1.ADDR_Bit := 7;
   Gas_Chanel_1_1.Filter_On.SP := 16#02;
   Gas_Chanel_1_1.Filter_Off.SP := 16#02;
   Gas_Chanel_1_2.Use.Inverse := TRUE;
   Gas_Chanel_1_2.Use.Indirect := TRUE;
   Gas_Chanel_1_2.ADDR_Byte := 1;
   Gas_Chanel_1_2.ADDR_Bit := 0;
   Gas_Chanel_1_2.Filter_On.SP := 16#02;
   Gas_Chanel_1_2.Filter_Off.SP := 16#02;
   Gas_Chanel_2_1.Use.Inverse := TRUE;
   Gas_Chanel_2_1.Use.Indirect := TRUE;
   Gas_Chanel_2_1.ADDR_Byte := 1;
   Gas_Chanel_2_1.ADDR_Bit := 1;
   Gas_Chanel_2_1.Filter_On.SP := 16#02;
   Gas_Chanel_2_1.Filter_Off.SP := 16#02;
   Gas_Chanel_2_2.Use.Inverse := TRUE;
   Gas_Chanel_2_2.Use.Indirect := TRUE;
   Gas_Chanel_2_2.ADDR_Byte := 1;
   Gas_Chanel_2_2.ADDR_Bit := 2;
   Gas_Chanel_2_2.Filter_On.SP := 16#02;
   Gas_Chanel_2_2.Filter_Off.SP := 16#02;
   ALS_1.Use.Inverse := FALSE;
   ALS_1.Use.Indirect := TRUE;
   ALS_1.ADDR_Byte := 2;
   ALS_1.ADDR_Bit := 0;
   ALS_1.Filter_On.SP := 16#02;
   ALS_1.Filter_Off.SP := 16#02;
   KC_1.Use.Inverse := FALSE;
   KC_1.Use.Indirect := TRUE;
   KC_1.ADDR_Byte := 1;
   KC_1.ADDR_Bit := 3;
   KC_1.Filter_On.SP := 16#02;
   KC_1.Filter_Off.SP := 16#02;
   KC_2.Use.Inverse := FALSE;
   KC_2.Use.Indirect := TRUE;
   KC_2.ADDR_Byte := 1;
   KC_2.ADDR_Bit := 4;
   KC_2.Filter_On.SP := 16#02;
   KC_2.Filter_Off.SP := 16#02;
   signal_10.Use.Inverse := TRUE;
   signal_10.Use.Indirect := TRUE;
   signal_10.ADDR_Byte := 2;
   signal_10.ADDR_Bit := 7;
   signal_10.Filter_On.SP := 16#02;
   signal_10.Filter_Off.SP := 16#02;
   signal_11.Use.Inverse := TRUE;
   signal_11.Use.Indirect := TRUE;
   signal_11.ADDR_Byte := 2;
   signal_11.ADDR_Bit := 5;
   signal_11.Filter_On.SP := 16#02;
   signal_11.Filter_Off.SP := 16#02;
   signal_12.Use.Inverse := TRUE;
   signal_12.Use.Indirect := TRUE;
   signal_12.ADDR_Byte := 2;
   signal_12.ADDR_Bit := 6;
   signal_12.Filter_On.SP := 16#02;
   signal_12.Filter_Off.SP := 16#02;
   signal_13.Use.Inverse := TRUE;
   signal_13.Use.Indirect := TRUE;
   signal_13.ADDR_Byte := 3;
   signal_13.ADDR_Bit := 0;
   signal_13.Filter_On.SP := 16#02;
   signal_13.Filter_Off.SP := 16#02;
END_DATA_BLOCK

DATA_BLOCK "DOx_1_DB"   // DB210
VERSION : 0.1
// stored: AutoNumber false, DBAccessibleFromOPCUA true, InstanceOfName DOx_1, InstanceOfType FB
"DOx_1"
BEGIN
   EZ_1_Alarm_Stop.Use.Inverse := TRUE;
   EZ_1_Alarm_Stop.Use.Indirect := TRUE;
   EZ_1_Alarm_Stop.Use.Impulse := FALSE;
   EZ_1_Alarm_Stop.ADDR_Byte := 0;
   EZ_1_Alarm_Stop.ADDR_Bit := 1;
   EZ_1_Alarm_Stop.T_Impulse.SP := 16#02;
   Red_Signal.Use.Inverse := FALSE;
   Red_Signal.Use.Indirect := TRUE;
   Red_Signal.Use.Impulse := FALSE;
   Red_Signal.ADDR_Byte := 0;
   Red_Signal.ADDR_Bit := 6;
   Red_Signal.T_Impulse.SP := 16#02;
   KC_1_Start.Use.Inverse := FALSE;
   KC_1_Start.Use.Indirect := TRUE;
   KC_1_Start.Use.Impulse := FALSE;
   KC_1_Start.ADDR_Byte := 0;
   KC_1_Start.ADDR_Bit := 4;
   KC_1_Start.T_Impulse.SP := 16#02;
   KC_2_Start.Use.Inverse := FALSE;
   KC_2_Start.Use.Indirect := TRUE;
   KC_2_Start.Use.Impulse := FALSE;
   KC_2_Start.ADDR_Byte := 0;
   KC_2_Start.ADDR_Bit := 5;
   KC_2_Start.T_Impulse.SP := 16#02;
   command_5.Use.Inverse := FALSE;
   command_5.Use.Indirect := TRUE;
   command_5.Use.Impulse := FALSE;
   command_5.ADDR_Byte := 0;
   command_5.ADDR_Bit := 9;
   command_5.T_Impulse.SP := 16#02;
   command_6.Use.Inverse := FALSE;
   command_6.Use.Indirect := TRUE;
   command_6.Use.Impulse := FALSE;
   command_6.ADDR_Byte := 0;
   command_6.ADDR_Bit := 9;
   command_6.T_Impulse.SP := 16#02;
   command_7.Use.Inverse := FALSE;
   command_7.Use.Indirect := TRUE;
   command_7.Use.Impulse := FALSE;
   command_7.ADDR_Byte := 0;
   command_7.ADDR_Bit := 9;
   command_7.T_Impulse.SP := 16#02;
   command_8.Use.Inverse := FALSE;
   command_8.Use.Indirect := TRUE;
   command_8.Use.Impulse := FALSE;
   command_8.ADDR_Byte := 0;
   command_8.ADDR_Bit := 9;
   command_8.T_Impulse.SP := 16#02;
   command_9.Use.Inverse := FALSE;
   command_9.Use.Indirect := TRUE;
   command_9.Use.Impulse := FALSE;
   command_9.ADDR_Byte := 0;
   command_9.ADDR_Bit := 9;
   command_9.T_Impulse.SP := 16#02;
   command_10.Use.Inverse := FALSE;
   command_10.Use.Indirect := TRUE;
   command_10.Use.Impulse := FALSE;
   command_10.ADDR_Byte := 0;
   command_10.ADDR_Bit := 9;
   command_10.T_Impulse.SP := 16#02;
   command_11.Use.Inverse := FALSE;
   command_11.Use.Indirect := TRUE;
   command_11.Use.Impulse := FALSE;
   command_11.ADDR_Byte := 0;
   command_11.ADDR_Bit := 9;
   command_11.T_Impulse.SP := 16#02;
   command_12.Use.Inverse := FALSE;
   command_12.Use.Indirect := TRUE;
   command_12.Use.Impulse := FALSE;
   command_12.ADDR_Byte := 0;
   command_12.ADDR_Bit := 9;
   command_12.T_Impulse.SP := 16#02;
END_DATA_BLOCK

DATA_BLOCK "Motors_DB"   // DB240
VERSION : 0.1
// stored: AutoNumber false, DBAccessibleFromOPCUA true, InstanceOfName Motors, InstanceOfType FB
"Motors"
BEGIN
END_DATA_BLOCK

DATA_BLOCK "PIDx_DB"   // DB260
VERSION : 0.1
// stored: AutoNumber false, DBAccessibleFromOPCUA true, InstanceOfName PIDx, InstanceOfType FB
"PIDx"
BEGIN
END_DATA_BLOCK

DATA_BLOCK "Valves_DB"   // DB250
VERSION : 0.1
// stored: AutoNumber false, DBAccessibleFromOPCUA true, InstanceOfName Valves, InstanceOfType FB
"Valves"
BEGIN
END_DATA_BLOCK

DATA_BLOCK "FB_DRV_Start_DB"   // DB100
VERSION : 0.1
// stored: AutoNumber false, DBAccessibleFromOPCUA true, InstanceOfName FB_DRV_Start, InstanceOfType FB
"FB_DRV_Start"
BEGIN
   x.Stat[0..10] := FALSE;
   x.ADD_D := 7;
   x.Min_D := 7;
   x.Time_D.SP_D := 4;
   x.Time_D.SP_H := 0;
   x.Time_D.SP_M := 0;
   x.Time_D.SP_S := 0;
END_DATA_BLOCK

DATA_BLOCK "Historian_DB"   // DB88
VERSION : 0.1
// stored: AutoNumber false, DBAccessibleFromOPCUA true, InstanceOfName Historian, InstanceOfType FB
"Historian"
BEGIN
END_DATA_BLOCK

DATA_BLOCK "Time_SYS_DB"   // DB95
VERSION : 0.1
// stored: AutoNumber false, DBAccessibleFromOPCUA true, InstanceOfName Time_SYS, InstanceOfType FB
"Time_SYS"
BEGIN
   TimeZone.Bias := 180;
   TimeZone.DaylightBias := 60;
   TimeZone.DaylightStartMonth := 3;
   TimeZone.DaylightStartWeek := 5;
   TimeZone.DaylightStartWeekday := 7;
   TimeZone.DaylightStartHour := 2;
   TimeZone.DaylightStartMinute := 0;
   TimeZone.StandardStartMonth := 10;
   TimeZone.StandardStartWeek := 5;
   TimeZone.StandardStartWeekday := 1;
   TimeZone.StandardStartHour := 3;
   TimeZone.StandardStartMinute := 0;
   TimeZone.TimeZoneName := 'GMT+3';
   SET_TIMEZONE.REQ := FALSE;
   SET_TIMEZONE.TimeZone.Bias := 180;
   SET_TIMEZONE.TimeZone.DaylightBias := 60;
   SET_TIMEZONE.TimeZone.DaylightStartMonth := 3;
   SET_TIMEZONE.TimeZone.DaylightStartWeek := 5;
   SET_TIMEZONE.TimeZone.DaylightStartWeekday := 7;
   SET_TIMEZONE.TimeZone.DaylightStartHour := 2;
   SET_TIMEZONE.TimeZone.DaylightStartMinute := 0;
   SET_TIMEZONE.TimeZone.StandardStartMonth := 10;
   SET_TIMEZONE.TimeZone.StandardStartWeek := 5;
   SET_TIMEZONE.TimeZone.StandardStartWeekday := 1;
   SET_TIMEZONE.TimeZone.StandardStartHour := 3;
   SET_TIMEZONE.TimeZone.StandardStartMinute := 0;
   SET_TIMEZONE.TimeZone.TimeZoneName := 'GMT+3';
   SET_TIMEZONE.DONE := FALSE;
   SET_TIMEZONE.BUSY := FALSE;
   SET_TIMEZONE.ERROR := FALSE;
   SET_TIMEZONE.STATUS := 16#7000;
END_DATA_BLOCK

DATA_BLOCK "LE_1_DB"   // DB300
VERSION : 0.1
// stored: AutoNumber false, DBAccessibleFromOPCUA true, InstanceOfName AI_ex, InstanceOfType FB
"AI_ex"
BEGIN
   Converter.Lim_High := FALSE;
   Converter.Lim_Low := FALSE;
   Converter.Inverse := FALSE;
   Converter.Min_In := 0.0;
   Converter.Min_Out := 0.0;
   Converter.Max_In := 4946.0;
   Converter.Max_Out := 100.0;
   Tx[0..1].SP := 3.0;
   Tx[2..5].SP := 1.0;
   Tx[0..5].One := 0.1;
END_DATA_BLOCK

DATA_BLOCK "TE_1_DB"   // DB301
VERSION : 0.1
// stored: AutoNumber false, DBAccessibleFromOPCUA true, InstanceOfName AI_ex, InstanceOfType FB
"AI_ex"
BEGIN
   Converter.Lim_High := FALSE;
   Converter.Lim_Low := FALSE;
   Converter.Inverse := FALSE;
   Converter.Min_In := 0.0;
   Converter.Min_Out := 0.0;
   Converter.Max_In := 27648.0;
   Converter.Max_Out := 100.0;
   Tx[0..1].SP := 3.0;
   Tx[2..5].SP := 1.0;
   Tx[0..5].One := 0.1;
END_DATA_BLOCK

DATA_BLOCK "AO_example_DB"   // DB400
VERSION : 0.1
// stored: AutoNumber false, DBAccessibleFromOPCUA true, InstanceOfName AO_ex, InstanceOfType FB
"AO_ex"
BEGIN
   Converter.Lim_High := FALSE;
   Converter.Lim_Low := FALSE;
   Converter.Inverse := FALSE;
   Converter.Min_In := 0.0;
   Converter.Min_Out := 0.0;
   Converter.Max_In := 0.0;
   Converter.Max_Out := 0.0;
   Slow.Use_Up := FALSE;
   Slow.Use_Down := FALSE;
   Slow.Step_Up := 0.125;
   Slow.Step_Down := 0.125;
   Slow.T_Up.SP := 1.0;
   Slow.T_Up.One := 0.1;
   Slow.T_Down.SP := 1.0;
   Slow.T_Down.One := 0.1;
END_DATA_BLOCK

DATA_BLOCK "ELZ_1_DB"   // DB500
VERSION : 0.1
// stored: AutoNumber false, DBAccessibleFromOPCUA true, InstanceOfName DRV_M_D_ELZ, InstanceOfType FB
"DRV_M_D_ELZ"
BEGIN
   Tx[0..1].SP := 2;
   Tx[2].SP := 20;
   Tx[3].SP := 10;
END_DATA_BLOCK

DATA_BLOCK "Pump_1_DB"   // DB600
VERSION : 0.1
// stored: AutoNumber false, DBAccessibleFromOPCUA true, InstanceOfName DRV_M_DA, InstanceOfType FB
"DRV_M_DA"
BEGIN
   Tx[0].SP := 2;
   Tx[1].SP := 5;
   Tx[2].SP := 15;
   Tx[3].SP := 2;
   Converter.Lim_High := FALSE;
   Converter.Lim_Low := FALSE;
   Converter.Inverse := FALSE;
   Converter.Min_In := 0.0;
   Converter.Min_Out := 0.0;
   Converter.Max_In := 200.0;
   Converter.Max_Out := 27648.0;
   Slow.Use_Up := FALSE;
   Slow.Use_Down := FALSE;
   Slow.Step_Up := 0.125;
   Slow.Step_Down := 0.125;
   Slow.T_Up.SP := 1.0;
   Slow.T_Up.One := 0.1;
   Slow.T_Down.SP := 1.0;
   Slow.T_Down.One := 0.1;
END_DATA_BLOCK

DATA_BLOCK "Pump_2_DB"   // DB601
VERSION : 0.1
// stored: AutoNumber false, DBAccessibleFromOPCUA true, InstanceOfName DRV_M_DA, InstanceOfType FB
"DRV_M_DA"
BEGIN
   Tx[0].SP := 2;
   Tx[1].SP := 5;
   Tx[2].SP := 15;
   Tx[3].SP := 2;
   Converter.Lim_High := FALSE;
   Converter.Lim_Low := FALSE;
   Converter.Inverse := FALSE;
   Converter.Min_In := 0.0;
   Converter.Min_Out := 0.0;
   Converter.Max_In := 120.0;
   Converter.Max_Out := 27648.0;
   Slow.Use_Up := FALSE;
   Slow.Use_Down := FALSE;
   Slow.Step_Up := 0.125;
   Slow.Step_Down := 0.125;
   Slow.T_Up.SP := 1.0;
   Slow.T_Up.One := 0.1;
   Slow.T_Down.SP := 1.0;
   Slow.T_Down.One := 0.1;
END_DATA_BLOCK

DATA_BLOCK "Pump_ELZ_DB"   // DB501
VERSION : 0.1
// stored: AutoNumber false, DBAccessibleFromOPCUA true, InstanceOfName DRV_M_D, InstanceOfType FB
"DRV_M_D"
BEGIN
   Tx[0..3].SP := 2;
END_DATA_BLOCK

DATA_BLOCK "PID_example_DB"   // DB900
VERSION : 0.1
// stored: AutoNumber false, DBAccessibleFromOPCUA true, InstanceOfName PID_ex, InstanceOfType FB
"PID_ex"
BEGIN
   CMD.Vector := FALSE;
   PID.IntegralResetMode := 4;
   PID.RunModeByStartup := TRUE;
   PID.SetSubstituteOutput := TRUE;
   PID.ActivateRecoverMode := TRUE;
   PID.CancelTuningLevel := 10.0;
   PID.SubstituteOutput := 0.0;
   PID.Config.InputPerOn := FALSE;
   PID.Config.InvertControl := FALSE;
   PID.Config.InputUpperLimit := 500.0;
   PID.Config.InputLowerLimit := -500.0;
   PID.Config.InputUpperWarning := 3.402822E+38;
   PID.Config.InputLowerWarning := -3.402822E+38;
   PID.Config.OutputUpperLimit := 100.0;
   PID.Config.OutputLowerLimit := 0.0;
   PID.Config.SetpointUpperLimit := 500.0;
   PID.Config.SetpointLowerLimit := -500.0;
   PID.Config.MinimumOnTime := 0.0;
   PID.Config.MinimumOffTime := 0.0;
   PID.Config.InputScaling.UpperPointIn := 27648.0;
   PID.Config.InputScaling.LowerPointIn := 0.0;
   PID.Config.InputScaling.UpperPointOut := 100.0;
   PID.Config.InputScaling.LowerPointOut := 0.0;
   PID.CycleTime.EnEstimation := TRUE;
   PID.CycleTime.EnMonitoring := TRUE;
   PID.CycleTime.Value := 0.2005371;
   PID.CtrlParamsBackUp.Gain := 1.0;
   PID.CtrlParamsBackUp.Ti := 20.0;
   PID.CtrlParamsBackUp.Td := 0.0;
   PID.CtrlParamsBackUp.TdFiltRatio := 0.2;
   PID.CtrlParamsBackUp.PWeighting := 1.0;
   PID.CtrlParamsBackUp.DWeighting := 1.0;
   PID.CtrlParamsBackUp.Cycle := 1.0;
   PID.PIDSelfTune.SUT.TuneRule := 1;
   PID.PIDSelfTune.TIR.TuneRule := 0;
   PID.Retain.CtrlParams.Gain := 1.5;
   PID.Retain.CtrlParams.Ti := 150.0;
   PID.Retain.CtrlParams.Td := 0.0;
   PID.Retain.CtrlParams.TdFiltRatio := 0.2;
   PID.Retain.CtrlParams.PWeighting := 1.0;
   PID.Retain.CtrlParams.DWeighting := 1.0;
   PID.Retain.CtrlParams.Cycle := 1.0;
   C.SP := 0.2;
   C.One := 0.1;
END_DATA_BLOCK

DATA_BLOCK "V_D2A_example_DB"   // DB800
VERSION : 0.1
// stored: AutoNumber false, DBAccessibleFromOPCUA true, InstanceOfName DRV_V_D2A, InstanceOfType FB
"DRV_V_D2A"
BEGIN
   Tx[0..4].SP := 2;
   Tx_Sm[0..2].SP := 16#02;
   Tx_R[0..1].SP := 1.0;
   Tx_R[0..1].One := 0.1;
END_DATA_BLOCK

DATA_BLOCK "V_D2_example_DB"   // DB700
VERSION : 0.1
// stored: AutoNumber false, DBAccessibleFromOPCUA true, InstanceOfName DRV_V_D2, InstanceOfType FB
"DRV_V_D2"
BEGIN
   Tx[0..4].SP := 2;
END_DATA_BLOCK

DATA_BLOCK "DB_Reset_All"   // DB1099
{ S7_Optimized_Access := 'TRUE' }
// stored: AutoNumber true, DBAccessibleFromOPCUA true, InstanceOfName IEC_TIMER, OfSystemLibElement IEC_TIMER, OfSystemLibVersion 1.0
"IEC_TIMER"
   // VAR
   //    PT : Time;
   //    ET { ExternalWritable := 'False'} : Time;
   //    IN : Bool;
   //    Q { ExternalWritable := 'False'} : Bool;
   // END_VAR
BEGIN
END_DATA_BLOCK

DATA_BLOCK "DB_pulse_01s"   // DB1100
{ S7_Optimized_Access := 'TRUE' }
// stored: AutoNumber true, DBAccessibleFromOPCUA true, InstanceOfName IEC_TIMER, OfSystemLibElement IEC_TIMER, OfSystemLibVersion 1.0
"IEC_TIMER"
   // VAR
   //    PT : Time;
   //    ET { ExternalWritable := 'False'} : Time;
   //    IN : Bool;
   //    Q { ExternalWritable := 'False'} : Bool;
   // END_VAR
BEGIN
END_DATA_BLOCK

DATA_BLOCK "DB_pulse_05s"   // DB1101
{ S7_Optimized_Access := 'TRUE' }
// stored: AutoNumber true, DBAccessibleFromOPCUA true, InstanceOfName IEC_TIMER, OfSystemLibElement IEC_TIMER, OfSystemLibVersion 1.0
"IEC_TIMER"
   // VAR
   //    PT : Time;
   //    ET { ExternalWritable := 'False'} : Time;
   //    IN : Bool;
   //    Q { ExternalWritable := 'False'} : Bool;
   // END_VAR
BEGIN
END_DATA_BLOCK

DATA_BLOCK "DB_pulse_10s"   // DB1104
{ S7_Optimized_Access := 'TRUE' }
// stored: AutoNumber true, DBAccessibleFromOPCUA true, InstanceOfName IEC_TIMER, OfSystemLibElement IEC_TIMER, OfSystemLibVersion 1.0
"IEC_TIMER"
   // VAR
   //    PT : Time;
   //    ET { ExternalWritable := 'False'} : Time;
   //    IN : Bool;
   //    Q { ExternalWritable := 'False'} : Bool;
   // END_VAR
BEGIN
END_DATA_BLOCK

DATA_BLOCK "DB_pulse_1m"   // DB1106
{ S7_Optimized_Access := 'TRUE' }
// stored: AutoNumber true, DBAccessibleFromOPCUA true, InstanceOfName IEC_TIMER, OfSystemLibElement IEC_TIMER, OfSystemLibVersion 1.0
"IEC_TIMER"
   // VAR
   //    PT : Time;
   //    ET { ExternalWritable := 'False'} : Time;
   //    IN : Bool;
   //    Q { ExternalWritable := 'False'} : Bool;
   // END_VAR
BEGIN
END_DATA_BLOCK

DATA_BLOCK "DB_pulse_1s"   // DB1102
{ S7_Optimized_Access := 'TRUE' }
// stored: AutoNumber true, DBAccessibleFromOPCUA true, InstanceOfName IEC_TIMER, OfSystemLibElement IEC_TIMER, OfSystemLibVersion 1.0
"IEC_TIMER"
   // VAR
   //    PT : Time;
   //    ET { ExternalWritable := 'False'} : Time;
   //    IN : Bool;
   //    Q { ExternalWritable := 'False'} : Bool;
   // END_VAR
BEGIN
END_DATA_BLOCK

DATA_BLOCK "DB_pulse_30s"   // DB1105
{ S7_Optimized_Access := 'TRUE' }
// stored: AutoNumber true, DBAccessibleFromOPCUA true, InstanceOfName IEC_TIMER, OfSystemLibElement IEC_TIMER, OfSystemLibVersion 1.0
"IEC_TIMER"
   // VAR
   //    PT : Time;
   //    ET { ExternalWritable := 'False'} : Time;
   //    IN : Bool;
   //    Q { ExternalWritable := 'False'} : Bool;
   // END_VAR
BEGIN
END_DATA_BLOCK

DATA_BLOCK "DB_pulse_5s"   // DB1103
{ S7_Optimized_Access := 'TRUE' }
// stored: AutoNumber true, DBAccessibleFromOPCUA true, InstanceOfName IEC_TIMER, OfSystemLibElement IEC_TIMER, OfSystemLibVersion 1.0
"IEC_TIMER"
   // VAR
   //    PT : Time;
   //    ET { ExternalWritable := 'False'} : Time;
   //    IN : Bool;
   //    Q { ExternalWritable := 'False'} : Bool;
   // END_VAR
BEGIN
END_DATA_BLOCK

DATA_BLOCK "MB_SERVER_DB"   // DB4
// stored: AutoNumber true, DBAccessibleFromOPCUA true, InstanceOfName MB_SERVER, OfSystemLibElement MB_SERVER, OfSystemLibVersion 5.2
"MB_SERVER"
   // VAR_INPUT
   //    DISCONNECT { ExternalVisible := 'False'} : Bool;
   // END_VAR
   // VAR_OUTPUT
   //    NDR { ExternalVisible := 'False'} : Bool;
   //    DR { ExternalVisible := 'False'} : Bool;
   //    ERROR { ExternalVisible := 'False'} : Bool;
   //    STATUS { ExternalVisible := 'False'} : Word;
   // END_VAR
   // VAR_IN_OUT
   //    MB_HOLD_REG : Variant;
   //    CONNECT : Variant;
   // END_VAR
   // VAR
   //    TCON { S7_SetPoint := 'True'} : TCON;
   //    TSEND { S7_SetPoint := 'True'} : TSEND;
   //    TRCV { S7_SetPoint := 'True'} : TRCV;
   //    TDIAG { S7_SetPoint := 'True'} : T_DIAG;
   //    TRESET { S7_SetPoint := 'True'} : T_RESET;
   //    TDISCON { S7_SetPoint := 'True'} : TDISCON;
   //    TDIAG_Status { S7_SetPoint := 'True'} : TDiag_Status;
   //    HR_Start_Offset : Word;
   //    QB_Start : UInt;
   //    QB_Count : UInt;
   //    QB_Read_Start : UInt;
   //    QB_Read_Count : UInt;
   //    IB_Read_Start : UInt;
   //    IB_Read_Count : UInt;
   //    Success_Count : Word;
   //    Request_Count : Word;
   //    Xmt_Rcv_Count : Word;
   //    Server_Message_Count : Word;
   //    Exception_Count : Word;
   //    Connected : Bool;
   //    Connection_ID { ExternalVisible := 'False'} : Word;
   //    MB_State : Word;
   //    TEMP_DATA { ExternalVisible := 'False'} : Array[0..262] of Byte;
   //    Data_Area_Array { S7_SetPoint := 'True'} : Array[1..8] of MB_DataArea;
   //    NDR_immediate : Bool;
   //    DR_immediate : Bool;
   //    BytesReceived : UDInt;
   // END_VAR
BEGIN
END_DATA_BLOCK
